C09134=1225.795,-112.726,-36.127,179.386,5.319,149.110
C09135=1225.800,-112.975,-36.117,179.383,5.319,149.111
C09136=1225.805,-113.226,-36.108,179.381,5.319,149.111
C09137=1225.810,-113.475,-36.097,179.379,5.318,149.112
C09138=1225.816,-113.725,-36.087,179.377,5.319,149.113
C09139=1225.821,-113.975,-36.077,179.374,5.318,149.113
C09140=1225.826,-114.224,-36.067,179.372,5.319,149.114
C09141=1225.831,-114.474,-36.057,179.369,5.318,149.115
C09142=1225.837,-114.724,-36.047,179.367,5.318,149.116
C09143=1225.842,-114.974,-36.037,179.365,5.318,149.116
C09144=1225.847,-115.224,-36.027,179.363,5.318,149.117
C09145=1225.853,-115.473,-36.017,179.360,5.318,149.117
C09146=1225.857,-115.723,-36.007,179.358,5.318,149.118
C09147=1225.863,-115.973,-35.997,179.356,5.318,149.119
C09148=1225.869,-116.223,-35.987,179.353,5.318,149.120
C09149=1225.873,-116.472,-35.978,179.351,5.318,149.120
C09150=1225.878,-116.722,-35.967,179.349,5.317,149.121
C09151=1225.884,-116.972,-35.957,179.347,5.318,149.122
C09152=1225.889,-117.221,-35.947,179.344,5.317,149.122
C09153=1225.895,-117.471,-35.938,179.342,5.318,149.123
C09154=1225.900,-117.721,-35.927,179.339,5.317,149.124
C09155=1225.905,-117.971,-35.917,179.337,5.318,149.124
C09156=1225.910,-118.220,-35.907,179.335,5.317,149.125
C09157=1225.915,-118.470,-35.898,179.333,5.317,149.126
C09158=1225.920,-118.720,-35.888,179.331,5.318,149.126
C09159=1225.926,-118.970,-35.878,179.328,5.317,149.127
C09160=1225.931,-119.219,-35.868,179.326,5.318,149.128
C09161=1225.937,-119.469,-35.858,179.323,5.317,149.128
C09162=1225.942,-119.718,-35.849,179.321,5.318,149.129
C09163=1225.947,-119.969,-35.838,179.319,5.317,149.130
C09164=1225.953,-120.219,-35.829,179.317,5.317,149.130
C09165=1225.957,-120.468,-35.819,179.314,5.317,149.131
C09166=1225.963,-120.718,-35.809,179.312,5.317,149.132
C09167=1225.968,-120.968,-35.800,179.310,5.317,149.133
C09168=1225.973,-121.218,-35.790,179.307,5.317,149.133
C09169=1225.978,-121.467,-35.780,179.306,5.317,149.134
C09170=1225.984,-121.717,-35.770,179.303,5.317,149.134
C09171=1225.989,-121.966,-35.761,179.301,5.317,149.135
C09172=1225.994,-122.216,-35.751,179.298,5.317,149.136
C09173=1226.000,-122.467,-35.741,179.296,5.317,149.137
C09174=1226.005,-122.716,-35.731,179.294,5.317,149.137
C09175=1226.010,-122.966,-35.721,179.292,5.317,149.138
C09176=1226.015,-123.215,-35.712,179.289,5.316,149.139
C09177=1226.021,-123.465,-35.702,179.287,5.317,149.139
C09178=1226.026,-123.716,-35.693,179.285,5.317,149.140
C09179=1226.031,-123.965,-35.682,179.282,5.317,149.141
C09180=1226.036,-124.214,-35.673,179.280,5.317,149.141
C09181=1226.042,-124.464,-35.663,179.278,5.316,149.142
C09182=1226.047,-124.714,-35.654,179.276,5.317,149.143
C09183=1226.053,-124.964,-35.644,179.273,5.316,149.143
C09184=1226.058,-125.213,-35.634,179.271,5.316,149.144
C09185=1226.063,-125.464,-35.625,179.269,5.316,149.145
C09186=1226.068,-125.713,-35.615,179.267,5.316,149.145
C09187=1226.074,-125.963,-35.606,179.264,5.316,149.146
C09188=1226.078,-126.213,-35.596,179.262,5.316,149.147
C09189=1225.657,-126.223,-35.632,179.258,5.320,149.149
C09190=1225.652,-125.973,-35.641,179.260,5.319,149.148
C09191=1225.646,-125.724,-35.651,179.263,5.320,149.147
C09192=1225.641,-125.474,-35.660,179.265,5.319,149.147
C09193=1225.636,-125.224,-35.671,179.267,5.320,149.146
C09194=1225.631,-124.975,-35.680,179.269,5.320,149.145
C09195=1225.625,-124.724,-35.690,179.272,5.320,149.145
C09196=1225.620,-124.475,-35.700,179.274,5.320,149.144
C09197=1225.614,-124.225,-35.709,179.276,5.320,149.143
C09198=1225.609,-123.976,-35.719,179.279,5.320,149.143
C09199=1225.603,-123.726,-35.728,179.281,5.319,149.142
C09200=1225.599,-123.476,-35.738,179.283,5.320,149.141
C09201=1225.594,-123.226,-35.748,179.285,5.320,149.141
C09202=1225.588,-122.976,-35.757,179.288,5.320,149.140
C09203=1225.583,-122.727,-35.767,179.290,5.320,149.139
C09204=1225.578,-122.477,-35.776,179.292,5.320,149.138
C09205=1225.572,-122.227,-35.787,179.294,5.320,149.138
C09206=1225.568,-121.977,-35.797,179.297,5.321,149.137
C09207=1225.562,-121.727,-35.806,179.299,5.320,149.137
C09208=1225.557,-121.478,-35.816,179.301,5.321,149.136
C09209=1225.551,-121.229,-35.826,179.304,5.320,149.135
C09210=1225.546,-120.979,-35.835,179.306,5.320,149.134
C09211=1225.541,-120.728,-35.845,179.308,5.321,149.134
C09212=1225.536,-120.479,-35.856,179.310,5.320,149.133
C09213=1225.531,-120.229,-35.864,179.313,5.321,149.132
C09214=1225.525,-119.979,-35.875,179.315,5.320,149.132
C09215=1225.520,-119.730,-35.884,179.317,5.321,149.131
C09216=1225.515,-119.479,-35.894,179.319,5.320,149.130
C09217=1225.510,-119.230,-35.904,179.322,5.321,149.130
C09218=1225.504,-118.981,-35.914,179.324,5.321,149.129
C09219=1225.499,-118.731,-35.924,179.326,5.320,149.128
C09220=1225.494,-118.481,-35.933,179.328,5.321,149.128
C09221=1225.489,-118.231,-35.944,179.331,5.320,149.127
C09222=1225.484,-117.982,-35.953,179.333,5.321,149.126
C09223=1225.478,-117.732,-35.963,179.335,5.321,149.126
C09224=1225.473,-117.481,-35.973,179.338,5.321,149.125
C09225=1225.468,-117.232,-35.983,179.340,5.321,149.124
C09226=1225.462,-116.983,-35.993,179.342,5.321,149.124
C09227=1225.457,-116.733,-36.003,179.344,5.321,149.123
C09228=1225.452,-116.482,-36.013,179.347,5.321,149.122
C09229=1225.447,-116.233,-36.023,179.349,5.321,149.122
C09230=1225.442,-115.984,-36.032,179.351,5.322,149.121
C09231=1225.436,-115.734,-36.043,179.353,5.321,149.120
C09232=1225.431,-115.484,-36.053,179.356,5.321,149.120
C09233=1225.426,-115.234,-36.062,179.358,5.322,149.119
C09234=1225.420,-114.985,-36.072,179.360,5.321,149.118
C09235=1225.415,-114.735,-36.083,179.363,5.322,149.117
C09236=1225.410,-114.485,-36.093,179.365,5.321,149.117
C09237=1225.405,-114.235,-36.103,179.367,5.322,149.116
C09238=1225.399,-113.985,-36.112,179.369,5.322,149.116
C09239=1225.394,-113.735,-36.123,179.372,5.322,149.115
C09240=1225.389,-113.486,-36.132,179.374,5.322,149.114
C09241=1225.384,-113.236,-36.143,179.377,5.322,149.113
C09242=1225.378,-112.987,-36.153,179.379,5.322,149.113
C09243=1225.374,-112.737,-36.163,179.382,5.322,149.112
C09244=1225.368,-112.487,-36.173,179.383,5.322,149.111
C09245=1225.362,-112.238,-36.183,179.385,5.322,149.111
C09246=1225.357,-111.987,-36.193,179.388,5.322,149.110
C09247=1225.352,-111.738,-36.203,179.390,5.322,149.109
C09248=1225.347,-111.488,-36.213,179.393,5.322,149.109
C09249=1225.342,-111.238,-36.223,179.395,5.322,149.108
C09250=1225.336,-110.988,-36.234,179.398,5.322,149.107
C09251=1225.331,-110.739,-36.243,179.399,5.322,149.107
C09252=1225.326,-110.489,-36.254,179.402,5.323,149.106
C09253=1225.321,-110.239,-36.264,179.404,5.322,149.105
C09254=1225.315,-109.990,-36.274,179.407,5.323,149.105
C09255=1225.311,-109.740,-36.284,179.409,5.322,149.104
C09256=1225.305,-109.490,-36.294,179.411,5.323,149.103
C09257=1225.300,-109.241,-36.305,179.413,5.323,149.102
C09258=1225.295,-108.990,-36.315,179.416,5.322,149.102
C09259=1225.289,-108.741,-36.325,179.418,5.323,149.101
C09260=1225.284,-108.492,-36.335,179.420,5.323,149.100
C09261=1225.279,-108.241,-36.346,179.422,5.323,149.100
C09262=1225.274,-107.992,-36.356,179.425,5.323,149.099
C09263=1225.268,-107.742,-36.366,179.427,5.323,149.098
C09264=1225.263,-107.492,-36.377,179.429,5.323,149.098
C09265=1225.258,-107.243,-36.386,179.432,5.323,149.097
C09266=1225.253,-106.993,-36.397,179.434,5.323,149.096
C09267=1225.247,-106.743,-36.407,179.436,5.324,149.096
C09268=1225.242,-106.494,-36.417,179.438,5.323,149.095
C09269=1225.237,-106.243,-36.428,179.441,5.324,149.094
C09270=1225.231,-105.994,-36.438,179.443,5.323,149.094
C09271=1225.226,-105.745,-36.448,179.446,5.324,149.093
C09272=1225.221,-105.494,-36.458,179.448,5.323,149.092
C09273=1225.216,-105.245,-36.468,179.451,5.324,149.091
C09274=1225.211,-104.995,-36.479,179.453,5.323,149.091
C09275=1225.205,-104.745,-36.489,179.455,5.323,149.090
C09276=1225.200,-104.496,-36.500,179.457,5.324,149.090
C09277=1225.195,-104.246,-36.511,179.459,5.323,149.089
C09278=1225.189,-103.996,-36.521,179.462,5.324,149.088
C09279=1225.185,-103.746,-36.531,179.464,5.324,149.087
C09280=1225.179,-103.497,-36.541,179.466,5.324,149.087
C09281=1225.174,-103.247,-36.552,179.469,5.324,149.086
C09282=1225.169,-102.997,-36.562,179.471,5.324,149.085
C09283=1225.163,-102.747,-36.572,179.473,5.324,149.085
C09284=1225.159,-102.498,-36.583,179.476,5.324,149.084
C09285=1225.153,-102.248,-36.594,179.478,5.324,149.083
C09286=1225.148,-101.998,-36.604,179.480,5.325,149.083
C09287=1225.142,-101.748,-36.614,179.482,5.324,149.082
C09288=1225.137,-101.498,-36.625,179.485,5.325,149.081
C09289=1225.133,-101.249,-36.635,179.487,5.324,149.080
C09290=1225.127,-100.978,-36.647,179.490,5.325,149.080
C09291=1225.121,-100.706,-36.658,179.492,5.324,149.079
C09292=1225.115,-100.436,-36.669,179.495,5.324,149.078
C09293=1225.110,-100.165,-36.681,179.498,5.325,149.077
C09294=1225.104,-99.915,-36.691,179.500,5.324,149.077
C09295=1225.099,-99.665,-36.702,179.503,5.325,149.076
C09296=1225.093,-99.416,-36.712,179.504,5.325,149.075
C09297=1225.089,-99.166,-36.723,179.507,5.325,149.075
C09298=1225.084,-98.917,-36.733,179.509,5.325,149.074
C09299=1225.079,-98.666,-36.744,179.512,5.325,149.073
C09300=1225.074,-98.418,-36.755,179.514,5.325,149.073
C09301=1225.069,-98.167,-36.765,179.516,5.325,149.072
C09302=1225.063,-97.918,-36.775,179.518,5.325,149.071
C09303=1225.058,-97.667,-36.786,179.521,5.325,149.070
C09304=1225.053,-97.419,-36.797,179.523,5.325,149.070
C09305=1225.047,-97.168,-36.808,179.525,5.325,149.069
C09306=1225.041,-96.918,-36.818,179.527,5.326,149.069
C09307=1225.037,-96.669,-36.830,179.530,5.325,149.068
C09308=1225.031,-96.419,-36.840,179.532,5.326,149.067
C09309=1225.026,-96.169,-36.850,179.534,5.325,149.066
C09310=1225.020,-95.919,-36.861,179.537,5.326,149.066
C09311=1225.016,-95.670,-36.872,179.539,5.325,149.065
C09312=1225.010,-95.420,-36.882,179.542,5.326,149.064
C09313=1225.005,-95.171,-36.893,179.544,5.326,149.064
C09314=1225.000,-94.921,-36.904,179.547,5.326,149.063
C09315=1224.995,-94.671,-36.914,179.549,5.326,149.062
C09316=1224.990,-94.421,-36.925,179.551,5.326,149.061
C09317=1224.985,-94.172,-36.936,179.553,5.326,149.061
C09318=1224.980,-93.921,-36.946,179.556,5.326,149.060
C09319=1224.974,-93.673,-36.957,179.558,5.326,149.060
C09320=1224.969,-93.422,-36.968,179.560,5.327,149.059
C09321=1224.963,-93.173,-36.979,179.562,5.326,149.058
C09322=1224.958,-92.923,-36.990,179.565,5.327,149.057
C09323=1224.953,-92.673,-37.000,179.567,5.326,149.057
C09324=1224.948,-92.424,-37.011,179.570,5.327,149.056
C09325=1224.943,-92.173,-37.022,179.572,5.326,149.055
C09326=1224.938,-91.924,-37.033,179.575,5.327,149.055
C09327=1224.933,-91.674,-37.043,179.577,5.326,149.054
C09328=1224.927,-91.425,-37.054,179.579,5.327,149.053
C09329=1224.922,-91.175,-37.065,179.582,5.327,149.052
C09330=1224.916,-90.926,-37.076,179.584,5.327,149.052
C09331=1224.911,-90.676,-37.087,179.586,5.327,149.051
C09332=1224.906,-90.425,-37.098,179.588,5.327,149.051
C09333=1224.901,-90.176,-37.108,179.591,5.327,149.050
C09334=1224.896,-89.926,-37.119,179.593,5.328,149.049
C09335=1224.891,-89.677,-37.130,179.595,5.327,149.048
C09336=1224.885,-89.427,-37.141,179.598,5.328,149.048
C09337=1224.880,-89.177,-37.152,179.600,5.327,149.047
C09338=1224.875,-88.928,-37.163,179.603,5.328,149.046
C09339=1224.870,-88.678,-37.174,179.605,5.327,149.046
C09340=1224.865,-88.428,-37.185,179.608,5.328,149.045
C09341=1224.860,-88.179,-37.195,179.610,5.327,149.044
C09342=1224.854,-87.929,-37.207,179.612,5.328,149.043
C09343=1224.849,-87.679,-37.217,179.614,5.328,149.043
C09344=1224.844,-87.430,-37.229,179.617,5.328,149.042
C09345=1224.839,-87.179,-37.239,179.619,5.328,149.041
C09346=1224.833,-86.930,-37.251,179.621,5.328,149.041
C09347=1224.828,-86.681,-37.262,179.623,5.328,149.040
C09348=1224.823,-86.430,-37.273,179.626,5.329,149.039
C09349=1224.818,-86.181,-37.284,179.628,5.328,149.039
C09350=1224.813,-85.931,-37.294,179.631,5.329,149.038
C09351=1224.808,-85.681,-37.306,179.633,5.328,149.037
C09352=1224.802,-85.432,-37.317,179.636,5.329,149.037
C09353=1224.797,-85.182,-37.328,179.638,5.328,149.036
C09354=1224.793,-84.932,-37.339,179.640,5.329,149.035
C09355=1224.786,-84.683,-37.350,179.642,5.328,149.034
C09356=1224.782,-84.433,-37.361,179.645,5.329,149.034
C09357=1224.777,-84.183,-37.372,179.647,5.329,149.033
C09358=1224.771,-83.934,-37.382,179.650,5.329,149.032
C09359=1224.766,-83.684,-37.394,179.652,5.329,149.032
C09360=1224.761,-83.434,-37.406,179.655,5.329,149.031
C09361=1224.756,-83.185,-37.416,179.657,5.329,149.030
C09362=1224.750,-82.935,-37.428,179.659,5.329,149.029
C09363=1224.745,-82.685,-37.439,179.662,5.329,149.029
C09364=1224.741,-82.435,-37.450,179.664,5.330,149.028
C09365=1224.734,-82.186,-37.461,179.666,5.330,149.028
C09366=1224.730,-81.936,-37.472,179.668,5.330,149.027
C09367=1224.725,-81.686,-37.484,179.671,5.330,149.026
C09368=1224.719,-81.436,-37.495,179.673,5.330,149.025
C09369=1224.714,-81.187,-37.506,179.676,5.330,149.025
C09370=1224.709,-80.937,-37.517,179.678,5.330,149.024
C09371=1224.704,-80.687,-37.529,179.681,5.330,149.023
C09372=1224.698,-80.438,-37.539,179.683,5.330,149.023
C09373=1224.694,-80.188,-37.550,179.685,5.330,149.022
C09374=1224.688,-79.938,-37.562,179.688,5.330,149.021
C09375=1224.683,-79.689,-37.573,179.690,5.331,149.020
C09376=1224.678,-79.440,-37.585,179.692,5.330,149.020
C09377=1224.672,-79.189,-37.596,179.695,5.331,149.019
C09378=1224.668,-78.939,-37.607,179.697,5.330,149.018
C09379=1224.663,-78.691,-37.618,179.700,5.331,149.018
C09380=1224.657,-78.441,-37.630,179.702,5.330,149.017
C09381=1224.652,-78.191,-37.641,179.704,5.331,149.016
C09382=1224.647,-77.940,-37.652,179.707,5.331,149.015
C09383=1224.642,-77.691,-37.664,179.709,5.331,149.015
C09384=1224.637,-77.442,-37.675,179.711,5.331,149.014
C09385=1224.631,-77.192,-37.686,179.713,5.331,149.014
C09386=1224.627,-76.942,-37.698,179.716,5.331,149.013
C09387=1224.621,-76.692,-37.710,179.718,5.332,149.012
C09388=1224.616,-76.443,-37.721,179.721,5.332,149.011
C09389=1224.610,-76.193,-37.732,179.723,5.332,149.011
C09390=1224.605,-75.943,-37.743,179.726,5.332,149.010
C09391=1224.600,-75.693,-37.755,179.728,5.332,149.009
C09392=1224.595,-75.444,-37.766,179.730,5.332,149.009
C09393=1224.590,-75.195,-37.777,179.733,5.332,149.008
C09394=1224.584,-74.924,-37.789,179.735,5.332,149.007
C09395=1224.579,-74.653,-37.802,179.738,5.332,149.006
C09396=1224.573,-74.383,-37.814,179.740,5.332,149.006
C09397=1224.568,-74.113,-37.827,179.743,5.333,149.005
C09398=1224.562,-73.863,-37.839,179.745,5.332,149.004
C09399=1224.557,-73.614,-37.850,179.748,5.333,149.003
C09400=1224.551,-73.364,-37.862,179.750,5.332,149.003
C09401=1224.547,-73.114,-37.873,179.753,5.333,149.002
C09402=1224.541,-72.864,-37.885,179.755,5.332,149.001
C09403=1224.537,-72.615,-37.896,179.757,5.333,149.001
C09404=1224.531,-72.365,-37.908,179.760,5.333,149.000
C09405=1224.526,-72.116,-37.919,179.762,5.333,148.999
C09406=1224.520,-71.866,-37.931,179.765,5.333,148.998
C09407=1224.516,-71.616,-37.942,179.767,5.333,148.998
C09408=1224.510,-71.366,-37.954,179.770,5.334,148.997
C09409=1224.506,-71.117,-37.965,179.772,5.333,148.996
C09410=1224.500,-70.867,-37.977,179.774,5.334,148.996
C09411=1224.495,-70.618,-37.988,179.776,5.333,148.995
C09412=1224.489,-70.368,-38.000,179.779,5.334,148.994
C09413=1224.485,-70.118,-38.011,179.781,5.334,148.994
C09414=1224.479,-69.868,-38.023,179.783,5.334,148.993
C09415=1224.474,-69.619,-38.035,179.785,5.334,148.992
C09416=1224.469,-69.369,-38.047,179.788,5.334,148.992
C09417=1224.464,-69.119,-38.058,179.791,5.335,148.991
C09418=1224.459,-68.869,-38.070,179.793,5.335,148.990
C09419=1224.453,-68.620,-38.081,179.796,5.335,148.989
C09420=1224.448,-68.370,-38.093,179.798,5.335,148.989
C09421=1224.443,-68.121,-38.104,179.800,5.335,148.988
C09422=1224.438,-67.871,-38.116,179.802,5.335,148.987
C09423=1224.433,-67.622,-38.128,179.805,5.335,148.987
C09424=1224.428,-67.372,-38.140,179.807,5.335,148.986
C09425=1224.422,-67.122,-38.152,179.810,5.335,148.985
C09426=1224.418,-66.872,-38.163,179.812,5.335,148.985
C09427=1224.412,-66.622,-38.175,179.815,5.335,148.984
C09428=1224.407,-66.373,-38.187,179.817,5.336,148.983
C09429=1224.401,-66.123,-38.198,179.819,5.336,148.982
C09430=1224.396,-65.874,-38.211,179.822,5.336,148.982
C09431=1224.392,-65.624,-38.222,179.824,5.336,148.981
C09432=1224.386,-65.374,-38.234,179.827,5.336,148.980
C09433=1224.381,-65.125,-38.246,179.829,5.336,148.980
C09434=1224.376,-64.875,-38.257,179.832,5.336,148.979
C09435=1224.371,-64.626,-38.270,179.834,5.336,148.978
C09436=1224.366,-64.376,-38.281,179.836,5.336,148.977
C09437=1224.361,-64.126,-38.293,179.839,5.337,148.977
C09438=1224.355,-63.876,-38.305,179.841,5.337,148.976
C09439=1224.350,-63.626,-38.317,179.844,5.337,148.975
C09440=1224.346,-63.377,-38.329,179.846,5.337,148.975
C09441=1224.340,-63.127,-38.340,179.848,5.337,148.974
C09442=1224.335,-62.877,-38.352,179.851,5.337,148.973
C09443=1224.329,-62.627,-38.364,179.853,5.337,148.973
C09444=1224.325,-62.378,-38.376,179.855,5.337,148.972
C09445=1224.319,-62.128,-38.388,179.858,5.337,148.971
C09446=1224.314,-61.878,-38.400,179.861,5.338,148.970
C09447=1224.309,-61.629,-38.411,179.863,5.337,148.970
C09448=1224.304,-61.379,-38.424,179.865,5.338,148.969
C09449=1224.299,-61.130,-38.436,179.867,5.338,148.968
C09450=1224.293,-60.880,-38.448,179.870,5.338,148.968
C09451=1224.289,-60.631,-38.460,179.872,5.338,148.967
C09452=1224.284,-60.381,-38.472,179.875,5.338,148.966
C09453=1224.278,-60.131,-38.483,179.878,5.339,148.965
C09454=1224.273,-59.881,-38.496,179.879,5.339,148.965
C09455=1224.268,-59.632,-38.507,179.882,5.339,148.964
C09456=1224.263,-59.382,-38.519,179.884,5.339,148.964
C09457=1224.258,-59.133,-38.532,179.887,5.339,148.963
C09458=1224.252,-58.883,-38.544,179.889,5.339,148.962
C09459=1224.247,-58.633,-38.556,179.891,5.339,148.961
C09460=1224.242,-58.384,-38.568,179.894,5.340,148.961
C09461=1224.237,-58.134,-38.579,179.896,5.340,148.960
C09462=1224.232,-57.884,-38.592,179.899,5.340,148.959
C09463=1224.227,-57.634,-38.604,179.901,5.340,148.959
C09464=1224.221,-57.385,-38.616,179.904,5.340,148.958
C09465=1224.217,-57.136,-38.628,179.906,5.340,148.957
C09466=1224.211,-56.886,-38.640,179.908,5.340,148.957
C09467=1224.206,-56.636,-38.652,179.911,5.341,148.956
C09468=1224.201,-56.386,-38.664,179.913,5.340,148.955
C09469=1224.196,-56.137,-38.677,179.916,5.341,148.954
C09470=1224.190,-55.887,-38.689,179.918,5.341,148.954
C09471=1224.186,-55.638,-38.701,179.920,5.341,148.953
C09472=1224.180,-55.388,-38.713,179.923,5.341,148.952
C09473=1224.175,-55.139,-38.725,179.925,5.341,148.952
C09474=1224.170,-54.888,-38.737,179.928,5.342,148.951
C09475=1224.165,-54.638,-38.749,179.930,5.341,148.950
C09476=1224.160,-54.389,-38.762,179.933,5.342,148.950
C09477=1224.154,-54.139,-38.774,179.935,5.341,148.949
C09478=1224.150,-53.890,-38.786,179.937,5.342,148.948
C09479=1224.145,-53.641,-38.798,179.939,5.342,148.947
C09480=1224.139,-53.391,-38.810,179.942,5.342,148.947
C09481=1224.134,-53.141,-38.823,179.945,5.343,148.946
C09482=1224.129,-52.891,-38.835,179.947,5.342,148.945
C09483=1224.124,-52.642,-38.847,179.950,5.343,148.945
C09484=1224.119,-52.392,-38.860,179.952,5.342,148.944
C09485=1224.114,-52.142,-38.872,179.954,5.343,148.943
C09486=1224.108,-51.892,-38.884,179.957,5.343,148.942
C09487=1224.103,-51.643,-38.897,179.959,5.343,148.942
C09488=1224.098,-51.394,-38.909,179.962,5.343,148.941
C09489=1224.093,-51.144,-38.921,179.964,5.343,148.940
C09490=1224.088,-50.895,-38.933,179.966,5.344,148.940
C09491=1224.083,-50.645,-38.945,179.969,5.344,148.939
C09492=1224.078,-50.395,-38.958,179.971,5.344,148.938
C09493=1224.073,-50.145,-38.971,179.974,5.344,148.938
C09494=1224.068,-49.895,-38.983,179.976,5.344,148.937
C09495=1224.063,-49.646,-38.995,179.979,5.344,148.936
C09496=1224.057,-49.396,-39.007,179.981,5.345,148.935
C09497=1224.052,-49.147,-39.020,179.983,5.345,148.935
C09498=1224.046,-48.877,-39.034,179.986,5.345,148.934
C09499=1224.041,-48.607,-39.047,179.989,5.345,148.933
C09500=1224.036,-48.337,-39.060,179.991,5.345,148.932
C09501=1224.030,-48.067,-39.073,179.994,5.345,148.932
C09502=1224.025,-47.818,-39.086,179.997,5.346,148.931
C09503=1224.020,-47.569,-39.098,179.999,5.345,148.930
C09504=1224.015,-47.319,-39.111,-179.999,5.346,148.930
C09505=1224.010,-47.069,-39.123,-179.997,5.346,148.929
C09506=1224.004,-46.819,-39.136,-179.994,5.346,148.928
C09507=1223.999,-46.570,-39.149,-179.991,5.347,148.927
C09508=1223.994,-46.320,-39.161,-179.989,5.346,148.927
C09509=1223.988,-46.070,-39.173,-179.986,5.347,148.926
C09510=1223.984,-45.820,-39.186,-179.984,5.346,148.925
C09511=1223.979,-45.571,-39.199,-179.982,5.347,148.925
C09512=1223.973,-45.321,-39.211,-179.979,5.347,148.924
C09513=1223.968,-45.072,-39.224,-179.977,5.347,148.923
C09514=1223.963,-44.822,-39.236,-179.974,5.347,148.923
C09515=1223.959,-44.572,-39.249,-179.972,5.347,148.922
C09516=1223.953,-44.322,-39.261,-179.970,5.348,148.921
C09517=1223.948,-44.073,-39.274,-179.967,5.348,148.920
C09518=1223.943,-43.824,-39.286,-179.965,5.348,148.920
C09519=1223.938,-43.575,-39.299,-179.962,5.348,148.919
C09520=1223.933,-43.324,-39.312,-179.960,5.348,148.918
C09521=1223.927,-43.075,-39.325,-179.957,5.348,148.918
C09522=1223.922,-42.825,-39.337,-179.955,5.349,148.917
C09523=1223.917,-42.576,-39.349,-179.953,5.349,148.916
C09524=1223.912,-42.326,-39.362,-179.950,5.349,148.916
C09525=1223.907,-42.076,-39.375,-179.947,5.350,148.915
C09526=1223.902,-41.827,-39.388,-179.945,5.349,148.914
C09527=1223.896,-41.577,-39.401,-179.943,5.350,148.913
C09528=1223.891,-41.327,-39.413,-179.940,5.349,148.913
C09529=1223.886,-41.077,-39.426,-179.938,5.350,148.912
C09530=1223.881,-40.828,-39.438,-179.935,5.350,148.911
C09531=1223.877,-40.578,-39.451,-179.933,5.350,148.911
C09532=1223.872,-40.329,-39.464,-179.930,5.350,148.910
C09533=1223.866,-40.079,-39.476,-179.928,5.351,148.909
C09534=1223.861,-39.830,-39.490,-179.926,5.351,148.909
C09535=1223.856,-39.580,-39.503,-179.923,5.351,148.908
C09536=1223.851,-39.330,-39.515,-179.921,5.351,148.907
C09537=1223.846,-39.081,-39.528,-179.918,5.351,148.906
C09538=1223.841,-38.831,-39.541,-179.916,5.352,148.906
C09539=1223.835,-38.581,-39.554,-179.913,5.351,148.905
C09540=1223.830,-38.332,-39.567,-179.911,5.352,148.904
C09541=1223.825,-38.083,-39.579,-179.909,5.352,148.904
C09542=1223.820,-37.832,-39.591,-179.906,5.352,148.903
C09543=1223.814,-37.583,-39.605,-179.903,5.353,148.902
C09544=1223.809,-37.333,-39.617,-179.901,5.352,148.902
C09545=1223.805,-37.083,-39.630,-179.899,5.353,148.901
C09546=1223.800,-36.834,-39.643,-179.896,5.353,148.900
C09547=1223.794,-36.584,-39.656,-179.894,5.353,148.899
C09548=1223.790,-36.335,-39.670,-179.891,5.353,148.899
C09549=1223.784,-36.086,-39.682,-179.889,5.354,148.898
C09550=1223.779,-35.836,-39.695,-179.887,5.354,148.897
C09551=1223.774,-35.586,-39.708,-179.884,5.354,148.897
C09552=1223.769,-35.337,-39.721,-179.882,5.354,148.896
C09553=1223.764,-35.087,-39.734,-179.879,5.354,148.895
C09554=1223.759,-34.837,-39.747,-179.876,5.355,148.895
C09555=1223.753,-34.588,-39.760,-179.874,5.354,148.894
C09556=1223.748,-34.338,-39.772,-179.872,5.355,148.893
C09557=1223.744,-34.088,-39.785,-179.869,5.355,148.892
C09558=1223.738,-33.839,-39.799,-179.867,5.355,148.892
C09559=1223.733,-33.589,-39.811,-179.864,5.356,148.891
C09560=1223.728,-33.339,-39.824,-179.862,5.356,148.890
C09561=1223.722,-33.090,-39.837,-179.860,5.356,148.890
C09562=1223.718,-32.840,-39.851,-179.857,5.356,148.889
C09563=1223.713,-32.591,-39.864,-179.855,5.356,148.888
C09564=1223.707,-32.341,-39.877,-179.852,5.356,148.888
C09565=1223.703,-32.091,-39.890,-179.849,5.357,148.887
C09566=1223.698,-31.842,-39.902,-179.847,5.357,148.886
C09567=1223.692,-31.592,-39.916,-179.845,5.357,148.885
C09568=1223.687,-31.342,-39.928,-179.842,5.358,148.885
C09569=1223.682,-31.094,-39.942,-179.840,5.357,148.884
C09570=1223.677,-30.843,-39.955,-179.837,5.358,148.883
C09571=1223.672,-30.594,-39.968,-179.835,5.358,148.883
C09572=1223.667,-30.344,-39.982,-179.833,5.358,148.882
C09573=1223.662,-30.094,-39.994,-179.830,5.358,148.881
C09574=1223.657,-29.846,-40.007,-179.827,5.359,148.881
C09575=1223.652,-29.595,-40.021,-179.825,5.359,148.880
C09576=1223.646,-29.346,-40.034,-179.823,5.359,148.879
C09577=1223.641,-29.096,-40.047,-179.820,5.360,148.878
C09578=1223.636,-28.847,-40.060,-179.818,5.359,148.878
C09579=1223.632,-28.597,-40.073,-179.815,5.360,148.877
C09580=1223.626,-28.347,-40.087,-179.812,5.360,148.876
C09581=1223.621,-28.098,-40.099,-179.810,5.360,148.876
C09582=1223.616,-27.848,-40.114,-179.808,5.360,148.875
C09583=1223.611,-27.599,-40.126,-179.806,5.360,148.874
C09584=1223.605,-27.349,-40.140,-179.803,5.361,148.874
C09585=1223.601,-27.100,-40.153,-179.800,5.361,148.873
C09586=1223.596,-26.850,-40.166,-179.798,5.361,148.872
C09587=1223.590,-26.600,-40.179,-179.796,5.361,148.872
C09588=1223.586,-26.350,-40.192,-179.793,5.362,148.871
C09589=1223.580,-26.101,-40.206,-179.791,5.361,148.870
C09590=1223.576,-25.851,-40.219,-179.788,5.362,148.869
C09591=1223.570,-25.602,-40.232,-179.786,5.362,148.869
C09592=1223.566,-25.352,-40.246,-179.783,5.362,148.868
C09593=1223.560,-25.103,-40.259,-179.781,5.363,148.867
C09594=1223.556,-24.853,-40.273,-179.778,5.363,148.867
C09595=1223.550,-24.604,-40.286,-179.777,5.363,148.866
C09596=1223.545,-24.354,-40.299,-179.774,5.364,148.865
C09597=1223.540,-24.105,-40.313,-179.771,5.364,148.865
C09598=1223.535,-23.855,-40.326,-179.769,5.364,148.864
C09599=1223.529,-23.605,-40.339,-179.766,5.364,148.863
C09600=1223.525,-23.356,-40.353,-179.764,5.365,148.863
C09601=1223.519,-23.106,-40.366,-179.762,5.365,148.862
C09602=1223.514,-22.837,-40.381,-179.759,5.365,148.861
C09603=1223.509,-22.567,-40.395,-179.756,5.365,148.860
C09604=1223.503,-22.298,-40.409,-179.753,5.366,148.860
C09605=1223.497,-22.029,-40.424,-179.751,5.366,148.859
C09606=1223.493,-21.779,-40.437,-179.749,5.366,148.858
C09607=1223.487,-21.530,-40.451,-179.746,5.366,148.858
C09608=1223.483,-21.280,-40.464,-179.743,5.367,148.857
C09609=1223.477,-21.031,-40.478,-179.741,5.367,148.856
C09610=1223.472,-20.780,-40.491,-179.738,5.367,148.856
C09611=1223.467,-20.532,-40.505,-179.736,5.368,148.855
C09612=1223.462,-20.281,-40.518,-179.734,5.367,148.854
C09613=1223.457,-20.033,-40.532,-179.731,5.368,148.853
C09614=1223.452,-19.782,-40.545,-179.728,5.368,148.853
C09615=1223.447,-19.533,-40.560,-179.726,5.369,148.852
C09616=1223.442,-19.283,-40.572,-179.724,5.368,148.851
C09617=1223.437,-19.033,-40.586,-179.721,5.369,148.851
C09618=1223.431,-18.784,-40.600,-179.718,5.369,148.850
C09619=1223.427,-18.534,-40.613,-179.716,5.369,148.849
C09620=1223.421,-18.285,-40.627,-179.714,5.370,148.849
C09621=1223.416,-18.035,-40.641,-179.711,5.370,148.848
C09622=1223.412,-17.786,-40.654,-179.709,5.370,148.847
C09623=1223.406,-17.536,-40.668,-179.706,5.370,148.846
C09624=1223.401,-17.287,-40.681,-179.704,5.371,148.846
C09625=1223.396,-17.038,-40.695,-179.701,5.371,148.845
C09626=1223.391,-16.787,-40.709,-179.699,5.371,148.844
C09627=1223.386,-16.538,-40.723,-179.696,5.372,148.844
C09628=1223.381,-16.288,-40.736,-179.693,5.372,148.843
C09629=1223.376,-16.039,-40.750,-179.691,5.372,148.842
C09630=1223.370,-15.790,-40.764,-179.689,5.372,148.842
C09631=1223.366,-15.540,-40.777,-179.686,5.373,148.841
C09632=1223.361,-15.290,-40.791,-179.684,5.372,148.840
C09633=1223.355,-15.041,-40.805,-179.681,5.373,148.840
C09634=1223.350,-14.791,-40.818,-179.679,5.373,148.839
C09635=1223.346,-14.541,-40.832,-179.677,5.373,148.838
C09636=1223.340,-14.292,-40.846,-179.674,5.374,148.837
C09637=1223.335,-14.042,-40.860,-179.671,5.374,148.837
C09638=1223.330,-13.792,-40.873,-179.669,5.375,148.836
C09639=1223.325,-13.543,-40.887,-179.667,5.374,148.835
C09640=1223.320,-13.293,-40.901,-179.664,5.375,148.835
C09641=1223.315,-13.043,-40.915,-179.661,5.375,148.834
C09642=1223.310,-12.795,-40.928,-179.659,5.375,148.833
C09643=1223.305,-12.545,-40.943,-179.657,5.376,148.833
C09644=1223.300,-12.295,-40.956,-179.654,5.376,148.832
C09645=1223.294,-12.046,-40.970,-179.651,5.377,148.831
C09646=1223.290,-11.796,-40.984,-179.649,5.376,148.831
C09647=1223.285,-11.546,-40.998,-179.646,5.377,148.830
C09648=1223.279,-11.297,-41.011,-179.644,5.377,148.829
C09649=1223.274,-11.047,-41.026,-179.642,5.377,148.828
C09650=1223.269,-10.797,-41.040,-179.639,5.378,148.828
C09651=1223.264,-10.549,-41.053,-179.636,5.378,148.827
C09652=1223.259,-10.299,-41.068,-179.634,5.379,148.826
C09653=1223.254,-10.049,-41.081,-179.632,5.378,148.826
C09654=1223.249,-9.800,-41.095,-179.629,5.379,148.825
C09655=1223.244,-9.550,-41.109,-179.626,5.379,148.824
C09656=1223.239,-9.301,-41.123,-179.624,5.379,148.824
C09657=1223.234,-9.051,-41.137,-179.622,5.380,148.823
C09658=1223.229,-8.802,-41.151,-179.619,5.380,148.822
C09659=1223.224,-8.552,-41.165,-179.616,5.381,148.822
C09660=1223.219,-8.302,-41.179,-179.614,5.380,148.821
C09661=1223.213,-8.053,-41.193,-179.612,5.381,148.820
C09662=1223.208,-7.803,-41.207,-179.609,5.381,148.819
C09663=1223.204,-7.554,-41.221,-179.607,5.381,148.819
C09664=1223.199,-7.304,-41.235,-179.604,5.381,148.818
C09665=1223.193,-7.055,-41.249,-179.602,5.382,148.817
C09666=1223.189,-6.805,-41.263,-179.599,5.383,148.817
C09667=1223.184,-6.556,-41.278,-179.597,5.382,148.816
C09668=1223.179,-6.306,-41.292,-179.594,5.383,148.815
C09669=1223.173,-6.057,-41.306,-179.592,5.384,148.815
C09670=1223.168,-5.807,-41.319,-179.589,5.384,148.814
C09671=1223.163,-5.557,-41.334,-179.587,5.384,148.813
C09672=1223.158,-5.307,-41.348,-179.585,5.384,148.813
C09673=1223.154,-5.058,-41.362,-179.582,5.385,148.812
C09674=1223.148,-4.809,-41.376,-179.579,5.385,148.811
C09675=1223.143,-4.559,-41.390,-179.577,5.385,148.811
C09676=1223.138,-4.309,-41.404,-179.575,5.386,148.810
C09677=1223.133,-4.060,-41.418,-179.572,5.386,148.809
C09678=1223.128,-3.811,-41.432,-179.570,5.386,148.809
C09679=1223.123,-3.561,-41.447,-179.567,5.386,148.808
C09680=1223.118,-3.311,-41.461,-179.565,5.387,148.807
C09681=1223.113,-3.061,-41.475,-179.562,5.387,148.807
C09682=1223.108,-2.812,-41.489,-179.560,5.387,148.806
C09683=1223.102,-2.563,-41.503,-179.557,5.388,148.805
C09684=1223.098,-2.314,-41.518,-179.555,5.388,148.804
C09685=1223.093,-2.064,-41.533,-179.552,5.389,148.804
C09686=1223.088,-1.814,-41.547,-179.550,5.388,148.803
C09687=1223.083,-1.564,-41.561,-179.547,5.389,148.802
C09688=1223.078,-1.315,-41.575,-179.544,5.389,148.802
C09689=1223.072,-1.066,-41.589,-179.542,5.390,148.801
C09690=1223.067,-0.816,-41.604,-179.540,5.390,148.800
C09691=1223.062,-0.566,-41.618,-179.537,5.390,148.800
C09692=1223.057,-0.317,-41.632,-179.534,5.391,148.799
C09693=1223.052,-0.067,-41.646,-179.532,5.391,148.798
C09694=1223.047,0.183,-41.661,-179.530,5.391,148.798
C09695=1223.042,0.431,-41.675,-179.527,5.391,148.797
C09696=1223.037,0.681,-41.690,-179.524,5.392,148.796
C09697=1223.032,0.931,-41.704,-179.522,5.392,148.796
C09698=1223.027,1.180,-41.718,-179.520,5.392,148.795
C09699=1223.022,1.430,-41.733,-179.517,5.393,148.794
C09700=1223.017,1.680,-41.747,-179.514,5.393,148.793
C09701=1223.012,1.929,-41.762,-179.512,5.394,148.793
C09702=1223.007,2.179,-41.777,-179.509,5.394,148.792
C09703=1223.002,2.428,-41.790,-179.507,5.394,148.791
C09704=1222.997,2.678,-41.805,-179.505,5.395,148.791
C09705=1222.992,2.927,-41.819,-179.502,5.395,148.790
C09706=1222.987,3.196,-41.835,-179.499,5.395,148.789
C09707=1222.981,3.465,-41.850,-179.496,5.396,148.789
C09708=1222.976,3.734,-41.867,-179.494,5.396,148.788
C09709=1222.970,4.003,-41.882,-179.492,5.396,148.787
C09710=1222.965,4.252,-41.897,-179.489,5.397,148.787
C09711=1222.961,4.502,-41.911,-179.486,5.397,148.786
C09712=1222.956,4.752,-41.925,-179.484,5.398,148.785
C09713=1222.950,5.001,-41.939,-179.481,5.398,148.785
C09714=1222.945,5.250,-41.955,-179.479,5.398,148.784
C09715=1222.940,5.500,-41.969,-179.476,5.399,148.783
C09716=1222.935,5.750,-41.983,-179.474,5.399,148.782
C09717=1222.930,5.999,-41.998,-179.471,5.400,148.782
C09718=1222.925,6.249,-42.013,-179.469,5.399,148.781
C09719=1222.920,6.498,-42.027,-179.466,5.400,148.780
C09720=1222.915,6.748,-42.042,-179.464,5.400,148.780
C09721=1222.910,6.997,-42.057,-179.461,5.401,148.779
C09722=1222.905,7.247,-42.071,-179.458,5.401,148.778
C09723=1222.900,7.496,-42.086,-179.456,5.401,148.778
C09724=1222.895,7.746,-42.100,-179.454,5.402,148.777
C09725=1222.890,7.996,-42.115,-179.451,5.402,148.776
C09726=1222.885,8.245,-42.130,-179.448,5.403,148.776
C09727=1222.880,8.495,-42.144,-179.446,5.402,148.775
C09728=1222.875,8.744,-42.159,-179.444,5.403,148.774
C09729=1222.870,8.994,-42.174,-179.441,5.404,148.774
C09730=1222.865,9.244,-42.189,-179.439,5.404,148.773
C09731=1222.860,9.493,-42.204,-179.436,5.405,148.772
C09732=1222.855,9.742,-42.218,-179.434,5.405,148.772
C09733=1222.850,9.992,-42.233,-179.431,5.405,148.771
C09734=1222.845,10.241,-42.248,-179.429,5.406,148.770
C09735=1222.840,10.491,-42.263,-179.426,5.406,148.770
C09736=1222.835,10.740,-42.277,-179.423,5.407,148.769
C09737=1222.830,10.990,-42.293,-179.421,5.406,148.768
C09738=1222.825,11.239,-42.307,-179.419,5.407,148.768
C09739=1222.820,11.488,-42.322,-179.416,5.407,148.767
C09740=1222.814,11.738,-42.337,-179.413,5.408,148.766
C09741=1222.810,11.988,-42.352,-179.411,5.408,148.766
C09742=1222.805,12.237,-42.366,-179.409,5.408,148.765
C09743=1222.799,12.487,-42.382,-179.406,5.409,148.764
C09744=1222.794,12.736,-42.396,-179.403,5.409,148.763
C09745=1222.790,12.985,-42.411,-179.401,5.410,148.763
C09746=1222.785,13.235,-42.425,-179.398,5.410,148.762
C09747=1222.779,13.485,-42.441,-179.396,5.410,148.761
C09748=1222.775,13.734,-42.455,-179.394,5.411,148.761
C09749=1222.769,13.984,-42.471,-179.391,5.411,148.760
C09750=1222.764,14.233,-42.485,-179.389,5.412,148.760
C09751=1222.760,14.483,-42.500,-179.386,5.413,148.759
C09752=1222.754,14.732,-42.515,-179.384,5.412,148.758
C09753=1222.749,14.982,-42.530,-179.381,5.413,148.758
C09754=1222.745,15.231,-42.545,-179.379,5.413,148.757
C09755=1222.739,15.481,-42.560,-179.376,5.414,148.756
C09756=1222.734,15.730,-42.575,-179.373,5.414,148.755
C09757=1222.729,15.979,-42.590,-179.371,5.415,148.755
C09758=1222.724,16.230,-42.605,-179.369,5.415,148.754
C09759=1222.720,16.479,-42.620,-179.366,5.415,148.753
C09760=1222.714,16.728,-42.635,-179.363,5.416,148.753
C09761=1222.709,16.978,-42.650,-179.361,5.416,148.752
C09762=1222.704,17.227,-42.665,-179.358,5.417,148.751
C09763=1222.699,17.476,-42.680,-179.356,5.416,148.751
C09764=1222.694,17.726,-42.694,-179.353,5.417,148.750
C09765=1222.689,17.975,-42.710,-179.351,5.418,148.750
C09766=1222.684,18.225,-42.725,-179.348,5.418,148.749
C09767=1222.679,18.475,-42.740,-179.346,5.419,148.748
C09768=1222.675,18.724,-42.755,-179.343,5.420,148.748
C09769=1222.669,18.974,-42.771,-179.341,5.419,148.747
C09770=1222.665,19.223,-42.786,-179.338,5.420,148.746
C09771=1222.659,19.473,-42.801,-179.336,5.420,148.745
C09772=1222.654,19.722,-42.816,-179.333,5.421,148.745
C09773=1222.649,19.971,-42.831,-179.330,5.421,148.744
C09774=1222.644,20.220,-42.846,-179.328,5.422,148.743
C09775=1222.639,20.471,-42.862,-179.326,5.422,148.743
C09776=1222.635,20.720,-42.877,-179.323,5.422,148.742
C09777=1222.629,20.970,-42.892,-179.320,5.423,148.741
C09778=1222.625,21.219,-42.907,-179.318,5.423,148.741
C09779=1222.619,21.469,-42.922,-179.315,5.424,148.740
C09780=1222.614,21.718,-42.937,-179.313,5.425,148.740
C09781=1222.609,21.967,-42.953,-179.311,5.424,148.739
C09782=1222.605,22.217,-42.968,-179.308,5.425,148.738
C09783=1222.599,22.466,-42.984,-179.306,5.425,148.738
C09784=1222.595,22.716,-42.999,-179.303,5.426,148.737
C09785=1222.589,22.966,-43.013,-179.300,5.427,148.736
C09786=1222.584,23.215,-43.028,-179.298,5.427,148.735
C09787=1222.580,23.465,-43.044,-179.295,5.428,148.735
C09788=1222.574,23.714,-43.060,-179.293,5.427,148.734
C09789=1222.570,23.963,-43.075,-179.290,5.428,148.733
C09790=1222.564,24.213,-43.091,-179.288,5.428,148.733
C09791=1222.560,24.462,-43.106,-179.285,5.429,148.732
C09792=1222.555,24.712,-43.121,-179.282,5.429,148.731
C09793=1222.550,24.961,-43.136,-179.280,5.430,148.731
C09794=1222.545,25.210,-43.152,-179.278,5.430,148.730
C09795=1222.539,25.460,-43.167,-179.276,5.431,148.730
C09796=1222.534,25.709,-43.182,-179.273,5.431,148.729
C09797=1222.530,25.960,-43.198,-179.270,5.432,148.728
C09798=1222.524,26.209,-43.213,-179.268,5.432,148.728
C09799=1222.520,26.458,-43.228,-179.265,5.433,148.727
C09800=1222.514,26.707,-43.244,-179.262,5.433,148.726
C09801=1222.510,26.957,-43.259,-179.260,5.434,148.726
C09802=1222.505,27.207,-43.275,-179.258,5.434,148.725
C09803=1222.499,27.456,-43.291,-179.255,5.434,148.724
C09804=1222.495,27.705,-43.306,-179.252,5.435,148.723
C09805=1222.490,27.955,-43.322,-179.250,5.436,148.723
C09806=1222.484,28.205,-43.337,-179.247,5.436,148.722
C09807=1222.480,28.454,-43.352,-179.245,5.437,148.722
C09808=1222.474,28.703,-43.368,-179.242,5.437,148.721
C09809=1222.470,28.953,-43.384,-179.240,5.437,148.720
C09810=1222.464,29.222,-43.401,-179.237,5.438,148.720
C09811=1222.459,29.490,-43.417,-179.235,5.438,148.719
C09812=1222.454,29.758,-43.434,-179.232,5.439,148.718
C09813=1222.448,30.027,-43.450,-179.228,5.440,148.717
C09814=1222.443,30.277,-43.467,-179.226,5.439,148.717
C09815=1222.439,30.526,-43.482,-179.224,5.440,148.716
C09816=1222.433,30.775,-43.498,-179.222,5.441,148.716
C09817=1222.428,31.025,-43.513,-179.219,5.441,148.715
C09818=1222.423,31.275,-43.529,-179.216,5.442,148.714
C09819=1222.419,31.524,-43.544,-179.214,5.442,148.714
C09820=1222.413,31.773,-43.560,-179.211,5.443,148.713
C09821=1222.408,32.024,-43.576,-179.208,5.444,148.712
C09822=1222.403,32.272,-43.592,-179.206,5.443,148.711
C09823=1222.399,32.521,-43.607,-179.204,5.444,148.711
C09824=1222.394,32.772,-43.623,-179.201,5.444,148.710
C09825=1222.388,33.021,-43.639,-179.199,5.445,148.710
C09826=1222.383,33.270,-43.654,-179.196,5.446,148.709
C09827=1222.379,33.520,-43.670,-179.194,5.446,148.708
C09828=1222.374,33.769,-43.686,-179.191,5.447,148.708
C09829=1222.369,34.018,-43.701,-179.188,5.447,148.707
C09830=1222.364,34.268,-43.717,-179.186,5.448,148.706
C09831=1222.358,34.518,-43.733,-179.184,5.448,148.706
C09832=1222.354,34.766,-43.749,-179.181,5.448,148.705
C09833=1222.349,35.016,-43.765,-179.178,5.449,148.704
C09834=1222.344,35.266,-43.780,-179.176,5.450,148.704
C09835=1222.339,35.516,-43.796,-179.174,5.450,148.703
C09836=1222.334,35.765,-43.812,-179.171,5.451,148.702
C09837=1222.329,36.014,-43.828,-179.168,5.451,148.702
C09838=1222.324,36.264,-43.844,-179.166,5.452,148.701
C09839=1222.319,36.513,-43.859,-179.163,5.452,148.700
C09840=1222.314,36.762,-43.875,-179.160,5.453,148.700
C09841=1222.309,37.012,-43.891,-179.158,5.453,148.699
C09842=1222.304,37.262,-43.907,-179.156,5.453,148.698
C09843=1222.299,37.511,-43.923,-179.153,5.454,148.698
C09844=1222.294,37.760,-43.939,-179.151,5.455,148.697
C09845=1222.289,38.010,-43.955,-179.148,5.455,148.697
C09846=1222.284,38.259,-43.971,-179.146,5.456,148.696
C09847=1222.279,38.509,-43.987,-179.143,5.456,148.695
C09848=1222.275,38.759,-44.002,-179.140,5.457,148.695
C09849=1222.270,39.007,-44.019,-179.138,5.458,148.694
C09850=1222.264,39.257,-44.034,-179.135,5.458,148.693
C09851=1222.260,39.506,-44.051,-179.132,5.459,148.693
C09852=1222.254,39.756,-44.066,-179.130,5.460,148.692
C09853=1222.250,40.006,-44.082,-179.128,5.459,148.691
C09854=1222.245,40.255,-44.099,-179.125,5.460,148.691
C09855=1222.240,40.505,-44.115,-179.123,5.460,148.690
C09856=1222.235,40.753,-44.131,-179.120,5.461,148.689
C09857=1222.230,41.004,-44.147,-179.118,5.461,148.689
C09858=1222.225,41.252,-44.163,-179.115,5.462,148.688
C09859=1222.219,41.502,-44.179,-179.112,5.463,148.687
C09860=1222.215,41.751,-44.195,-179.110,5.464,148.687
C09861=1222.210,42.001,-44.211,-179.108,5.464,148.686
C09862=1222.205,42.251,-44.227,-179.105,5.465,148.686
C09863=1222.200,42.499,-44.243,-179.102,5.465,148.685
C09864=1222.195,42.750,-44.259,-179.100,5.466,148.684
C09865=1222.190,42.998,-44.276,-179.097,5.466,148.684
C09866=1222.185,43.248,-44.292,-179.094,5.467,148.683
C09867=1222.180,43.497,-44.308,-179.092,5.467,148.682
C09868=1222.175,43.747,-44.324,-179.090,5.467,148.682
C09869=1222.170,43.996,-44.340,-179.087,5.468,148.681
C09870=1222.166,44.246,-44.357,-179.085,5.469,148.680
C09871=1222.160,44.495,-44.372,-179.082,5.469,148.680
C09872=1222.156,44.744,-44.389,-179.080,5.470,148.679
C09873=1222.150,44.994,-44.405,-179.077,5.470,148.678
C09874=1222.146,45.243,-44.421,-179.074,5.471,148.678
C09875=1222.141,45.492,-44.438,-179.072,5.472,148.677
C09876=1222.135,45.743,-44.454,-179.069,5.472,148.677
C09877=1222.130,45.991,-44.470,-179.067,5.473,148.676
C09878=1222.125,46.241,-44.486,-179.064,5.473,148.675
C09879=1222.120,46.490,-44.503,-179.062,5.474,148.675
C09880=1222.116,46.740,-44.519,-179.059,5.475,148.674
C09881=1222.111,46.990,-44.535,-179.056,5.475,148.673
C09882=1222.106,47.239,-44.552,-179.054,5.476,148.673
C09883=1222.102,47.488,-44.568,-179.052,5.477,148.672
C09884=1222.096,47.738,-44.584,-179.049,5.477,148.672
C09885=1222.092,47.987,-44.601,-179.046,5.478,148.671
C09886=1222.086,48.236,-44.617,-179.044,5.477,148.670
C09887=1222.081,48.486,-44.633,-179.042,5.478,148.670
C09888=1222.076,48.735,-44.650,-179.039,5.479,148.669
C09889=1222.071,48.984,-44.666,-179.037,5.479,148.668
C09890=1222.067,49.235,-44.682,-179.034,5.480,148.668
C09891=1222.062,49.483,-44.699,-179.031,5.481,148.667
C09892=1222.056,49.733,-44.716,-179.029,5.481,148.666
C09893=1222.051,49.982,-44.732,-179.026,5.482,148.666
C09894=1222.047,50.232,-44.748,-179.024,5.482,148.665
C09895=1222.042,50.482,-44.765,-179.021,5.483,148.664
C09896=1222.037,50.730,-44.781,-179.019,5.484,148.664
C09897=1222.032,50.980,-44.798,-179.016,5.484,148.663
C09898=1222.026,51.229,-44.814,-179.014,5.485,148.663
C09899=1222.022,51.479,-44.831,-179.011,5.485,148.662
C09900=1222.017,51.728,-44.847,-179.008,5.486,148.661
C09901=1222.012,51.977,-44.864,-179.006,5.487,148.661
C09902=1222.007,52.227,-44.881,-179.003,5.487,148.660
C09903=1222.003,52.477,-44.898,-179.001,5.488,148.660
C09904=1221.997,52.726,-44.913,-178.998,5.489,148.659
C09905=1221.993,52.975,-44.930,-178.996,5.489,148.658
C09906=1221.988,53.224,-44.946,-178.993,5.490,148.657
C09907=1221.982,53.474,-44.963,-178.990,5.490,148.657
C09908=1221.978,53.723,-44.980,-178.988,5.491,148.656
C09909=1221.973,53.972,-44.996,-178.985,5.492,148.656
C09910=1221.968,54.222,-45.014,-178.983,5.492,148.655
C09911=1221.963,54.472,-45.030,-178.980,5.493,148.654
C09912=1221.958,54.721,-45.046,-178.978,5.493,148.654
C09913=1221.953,54.970,-45.063,-178.975,5.494,148.653
C09914=1221.947,55.239,-45.081,-178.972,5.495,148.652
C09915=1221.943,55.507,-45.099,-178.970,5.495,148.652
C09916=1221.937,55.775,-45.117,-178.967,5.496,148.651
C09917=1221.932,56.045,-45.135,-178.964,5.496,148.650
C09918=1221.927,56.294,-45.151,-178.962,5.497,148.650
C09919=1221.921,56.543,-45.168,-178.960,5.498,148.649
C09920=1221.917,56.793,-45.185,-178.957,5.498,148.649
C09921=1221.912,57.042,-45.202,-178.954,5.499,148.648
C09922=1221.907,57.291,-45.218,-178.952,5.499,148.647
C09923=1221.902,57.541,-45.235,-178.949,5.500,148.647
C09924=1221.898,57.790,-45.252,-178.946,5.501,148.646
C09925=1221.892,58.039,-45.269,-178.944,5.502,148.646
C09926=1221.887,58.289,-45.285,-178.942,5.502,148.645
C09927=1221.883,58.538,-45.302,-178.939,5.503,148.644
C09928=1221.878,58.788,-45.319,-178.936,5.503,148.644
C09929=1221.873,59.037,-45.336,-178.934,5.504,148.643
C09930=1221.867,59.287,-45.353,-178.932,5.505,148.642
C09931=1221.863,59.535,-45.370,-178.929,5.505,148.642
C09932=1221.859,59.785,-45.387,-178.926,5.506,148.641
C09933=1221.853,60.034,-45.404,-178.924,5.506,148.640
C09934=1221.848,60.283,-45.420,-178.921,5.507,148.640
C09935=1221.843,60.533,-45.438,-178.919,5.508,148.639
C09936=1221.839,60.783,-45.454,-178.916,5.509,148.639
C09937=1221.833,61.032,-45.471,-178.913,5.510,148.638
C09938=1221.828,61.281,-45.488,-178.910,5.510,148.637
C09939=1221.823,61.531,-45.505,-178.908,5.511,148.637
C09940=1221.819,61.780,-45.523,-178.905,5.512,148.636
C09941=1221.814,62.029,-45.539,-178.903,5.513,148.636
C09942=1221.809,62.279,-45.556,-178.900,5.513,148.635
C09943=1221.804,62.528,-45.573,-178.898,5.514,148.634
C09944=1221.799,62.778,-45.590,-178.895,5.514,148.634
C09945=1221.794,63.027,-45.606,-178.893,5.515,148.633
C09946=1221.789,63.276,-45.624,-178.890,5.516,148.632
C09947=1221.785,63.525,-45.641,-178.888,5.516,148.632
C09948=1221.779,63.775,-45.658,-178.885,5.517,148.631
C09949=1221.775,64.025,-45.675,-178.883,5.517,148.630
C09950=1221.770,64.274,-45.692,-178.880,5.518,148.630
C09951=1221.765,64.523,-45.709,-178.878,5.519,148.629
C09952=1221.760,64.772,-45.727,-178.875,5.520,148.629
C09953=1221.755,65.022,-45.743,-178.872,5.520,148.628
C09954=1221.750,65.272,-45.761,-178.870,5.521,148.627
C09955=1221.745,65.521,-45.778,-178.868,5.522,148.627
C09956=1221.740,65.770,-45.795,-178.865,5.522,148.626
C09957=1221.735,66.019,-45.812,-178.862,5.523,148.626
C09958=1221.731,66.268,-45.829,-178.860,5.523,148.625
C09959=1221.725,66.518,-45.847,-178.857,5.524,148.624
C09960=1221.721,66.768,-45.863,-178.855,5.525,148.624
C09961=1221.716,67.017,-45.881,-178.852,5.525,148.623
C09962=1221.711,67.266,-45.899,-178.850,5.526,148.623
C09963=1221.706,67.515,-45.915,-178.847,5.527,148.622
C09964=1221.701,67.764,-45.933,-178.845,5.527,148.621
C09965=1221.696,68.014,-45.950,-178.842,5.529,148.621
C09966=1221.691,68.264,-45.967,-178.839,5.529,148.620
C09967=1221.686,68.513,-45.985,-178.837,5.530,148.619
C09968=1221.682,68.762,-46.001,-178.834,5.531,148.619
C09969=1221.676,69.012,-46.019,-178.832,5.532,148.618
C09970=1221.672,69.261,-46.036,-178.829,5.532,148.618
C09971=1221.666,69.510,-46.053,-178.827,5.533,148.617
C09972=1221.662,69.759,-46.071,-178.824,5.533,148.616
C09973=1221.657,70.009,-46.088,-178.821,5.534,148.616
C09974=1221.652,70.258,-46.106,-178.819,5.535,148.615
C09975=1221.647,70.508,-46.123,-178.817,5.535,148.615
C09976=1221.642,70.757,-46.140,-178.814,5.536,148.614
C09977=1221.638,71.006,-46.158,-178.811,5.537,148.613
C09978=1221.632,71.256,-46.175,-178.809,5.537,148.613
C09979=1221.628,71.505,-46.192,-178.806,5.538,148.612
C09980=1221.623,71.755,-46.209,-178.803,5.539,148.612
C09981=1221.618,72.004,-46.227,-178.801,5.540,148.611
C09982=1221.613,72.253,-46.244,-178.799,5.541,148.610
C09983=1221.608,72.502,-46.262,-178.796,5.542,148.610
C09984=1221.603,72.752,-46.279,-178.793,5.542,148.609
C09985=1221.598,73.001,-46.297,-178.791,5.543,148.609
C09986=1221.593,73.250,-46.314,-178.789,5.544,148.608
C09987=1221.589,73.500,-46.332,-178.786,5.544,148.607
C09988=1221.584,73.749,-46.350,-178.783,5.545,148.607
C09989=1221.578,73.999,-46.367,-178.781,5.545,148.606
C09990=1221.574,74.247,-46.384,-178.778,5.546,148.605
C09991=1221.569,74.497,-46.402,-178.776,5.547,148.605
C09992=1221.564,74.746,-46.420,-178.773,5.547,148.604
C09993=1221.559,74.996,-46.437,-178.770,5.549,148.604
C09994=1221.555,75.245,-46.454,-178.767,5.549,148.603
C09995=1221.550,75.494,-46.472,-178.765,5.550,148.603
C09996=1221.545,75.744,-46.489,-178.763,5.551,148.602
//INST
///DATE 2021/06/15 17:22
///ATTR SC,RW,RJ
////FRAME ROBOT
///GROUP1 RB1
NOP
MOVL C00000 V=800.0 PL=0
MOVL C00001 V=800.0 PL=0
MOVL C00002 V=800.0 PL=0
MOVL C00003 V=800.0 PL=0
MOVL C00004 V=800.0 PL=0
MOVL C00005 V=800.0 PL=0
MOVL C00006 V=800.0 PL=0
MOVL C00007 V=800.0 PL=0
MOVL C00008 V=800.0 PL=0
MOVL C00009 V=800.0 PL=0
MOVL C00010 V=800.0 PL=0
MOVL C00011 V=800.0 PL=0
MOVL C00012 V=800.0 PL=0
MOVL C00013 V=800.0 PL=0
MOVL C00014 V=800.0 PL=0
MOVL C00015 V=800.0 PL=0
MOVL C00016 V=800.0 PL=0
MOVL C00017 V=800.0 PL=0
MOVL C00018 V=800.0 PL=0
MOVL C00019 V=800.0 PL=0
MOVL C00020 V=800.0 PL=0
MOVL C00021 V=800.0 PL=0
MOVL C00022 V=800.0 PL=0
MOVL C00023 V=800.0 PL=0
MOVL C00024 V=800.0 PL=0
MOVL C00025 V=800.0 PL=0
MOVL C00026 V=800.0 PL=0
MOVL C00027 V=800.0 PL=0
MOVL C00028 V=800.0 PL=0
MOVL C00029 V=800.0 PL=0
MOVL C00030 V=800.0 PL=0
MOVL C00031 V=800.0 PL=0
MOVL C00032 V=800.0 PL=0
MOVL C00033 V=800.0 PL=0
MOVL C00034 V=800.0 PL=0
MOVL C00035 V=800.0 PL=0
MOVL C00036 V=800.0 PL=0
MOVL C00037 V=800.0 PL=0
MOVL C00038 V=800.0 PL=0
MOVL C00039 V=800.0 PL=0
MOVL C00040 V=800.0 PL=0
MOVL C00041 V=800.0 PL=0
MOVL C00042 V=800.0 PL=0
MOVL C00043 V=800.0 PL=0
MOVL C00044 V=800.0 PL=0
MOVL C00045 V=800.0 PL=0
MOVL C00046 V=800.0 PL=0
MOVL C00047 V=800.0 PL=0
MOVL C00048 V=800.0 PL=0
MOVL C00049 V=800.0 PL=0
MOVL C00050 V=800.0 PL=0
MOVL C00051 V=800.0 PL=0
MOVL C00052 V=800.0 PL=0
MOVL C00053 V=800.0 PL=0
MOVL C00054 V=800.0 PL=0
MOVL C00055 V=800.0 PL=0
MOVL C00056 V=800.0 PL=0
MOVL C00057 V=800.0 PL=0
MOVL C00058 V=800.0 PL=0
MOVL C00059 V=800.0 PL=0
MOVL C00060 V=800.0 PL=0
MOVL C00061 V=800.0 PL=0
MOVL C00062 V=800.0 PL=0
MOVL C00063 V=800.0 PL=0
MOVL C00064 V=800.0 PL=0
MOVL C00065 V=800.0 PL=0
MOVL C00066 V=800.0 PL=0
MOVL C00067 V=800.0 PL=0
MOVL C00068 V=800.0 PL=0
MOVL C00069 V=800.0 PL=0
MOVL C00070 V=800.0 PL=0
MOVL C00071 V=800.0 PL=0
MOVL C00072 V=800.0 PL=0
MOVL C00073 V=800.0 PL=0
MOVL C00074 V=800.0 PL=0
MOVL C00075 V=800.0 PL=0
MOVL C00076 V=800.0 PL=0
MOVL C00077 V=800.0 PL=0
MOVL C00078 V=800.0 PL=0
MOVL C00079 V=800.0 PL=0
MOVL C00080 V=800.0 PL=0
MOVL C00081 V=800.0 PL=0
MOVL C00082 V=800.0 PL=0
MOVL C00083 V=800.0 PL=0
MOVL C00084 V=800.0 PL=0
MOVL C00085 V=800.0 PL=0
MOVL C00086 V=800.0 PL=0
MOVL C00087 V=800.0 PL=0
MOVL C00088 V=800.0 PL=0
MOVL C00089 V=800.0 PL=0
MOVL C00090 V=800.0 PL=0
MOVL C00091 V=800.0 PL=0
MOVL C00092 V=800.0 PL=0
MOVL C00093 V=800.0 PL=0
MOVL C00094 V=800.0 PL=0
MOVL C00095 V=800.0 PL=0
MOVL C00096 V=800.0 PL=0
MOVL C00097 V=800.0 PL=0
MOVL C00098 V=800.0 PL=0
MOVL C00099 V=800.0 PL=0
MOVL C00100 V=800.0 PL=0
MOVL C00101 V=800.0 PL=0
MOVL C00102 V=800.0 PL=0
MOVL C00103 V=800.0 PL=0
MOVL C00104 V=800.0 PL=0
MOVL C00105 V=800.0 PL=0
MOVL C00106 V=800.0 PL=0
MOVL C00107 V=800.0 PL=0
MOVL C00108 V=800.0 PL=0
MOVL C00109 V=800.0 PL=0
MOVL C00110 V=800.0 PL=0
MOVL C00111 V=800.0 PL=0
MOVL C00112 V=800.0 PL=0
MOVL C00113 V=800.0 PL=0
MOVL C00114 V=800.0 PL=0
MOVL C00115 V=800.0 PL=0
MOVL C00116 V=800.0 PL=0
MOVL C00117 V=800.0 PL=0
MOVL C00118 V=800.0 PL=0
MOVL C00119 V=800.0 PL=0
MOVL C00120 V=800.0 PL=0
MOVL C00121 V=800.0 PL=0
MOVL C00122 V=800.0 PL=0
MOVL C00123 V=800.0 PL=0
MOVL C00124 V=800.0 PL=0
MOVL C00125 V=800.0 PL=0
MOVL C00126 V=800.0 PL=0
MOVL C00127 V=800.0 PL=0
MOVL C00128 V=800.0 PL=0
MOVL C00129 V=800.0 PL=0
MOVL C00130 V=800.0 PL=0
MOVL C00131 V=800.0 PL=0
MOVL C00132 V=800.0 PL=0
MOVL C00133 V=800.0 PL=0
MOVL C00134 V=800.0 PL=0
MOVL C00135 V=800.0 PL=0
MOVL C00136 V=800.0 PL=0
MOVL C00137 V=800.0 PL=0
MOVL C00138 V=800.0 PL=0
MOVL C00139 V=800.0 PL=0
MOVL C00140 V=800.0 PL=0
MOVL C00141 V=800.0 PL=0
MOVL C00142 V=800.0 PL=0
MOVL C00143 V=800.0 PL=0
MOVL C00144 V=800.0 PL=0
MOVL C00145 V=800.0 PL=0
MOVL C00146 V=800.0 PL=0
MOVL C00147 V=800.0 PL=0
MOVL C00148 V=800.0 PL=0
MOVL C00149 V=800.0 PL=0
MOVL C00150 V=800.0 PL=0
MOVL C00151 V=800.0 PL=0
MOVL C00152 V=800.0 PL=0
MOVL C00153 V=800.0 PL=0
MOVL C00154 V=800.0 PL=0
MOVL C00155 V=800.0 PL=0
MOVL C00156 V=800.0 PL=0
MOVL C00157 V=800.0 PL=0
MOVL C00158 V=800.0 PL=0
MOVL C00159 V=800.0 PL=0
MOVL C00160 V=800.0 PL=0
MOVL C00161 V=800.0 PL=0
MOVL C00162 V=800.0 PL=0
MOVL C00163 V=800.0 PL=0
MOVL C00164 V=800.0 PL=0
MOVL C00165 V=800.0 PL=0
MOVL C00166 V=800.0 PL=0
MOVL C00167 V=800.0 PL=0
MOVL C00168 V=800.0 PL=0
MOVL C00169 V=800.0 PL=0
MOVL C00170 V=800.0 PL=0
MOVL C00171 V=800.0 PL=0
MOVL C00172 V=800.0 PL=0
MOVL C00173 V=800.0 PL=0
MOVL C00174 V=800.0 PL=0
MOVL C00175 V=800.0 PL=0
MOVL C00176 V=800.0 PL=0
MOVL C00177 V=800.0 PL=0
MOVL C00178 V=800.0 PL=0
MOVL C00179 V=800.0 PL=0
MOVL C00180 V=800.0 PL=0
MOVL C00181 V=800.0 PL=0
MOVL C00182 V=800.0 PL=0
MOVL C00183 V=800.0 PL=0
MOVL C00184 V=800.0 PL=0
MOVL C00185 V=800.0 PL=0
MOVL C00186 V=800.0 PL=0
MOVL C00187 V=800.0 PL=0
MOVL C00188 V=800.0 PL=0
MOVL C00189 V=800.0 PL=0
MOVL C00190 V=800.0 PL=0
MOVL C00191 V=800.0 PL=0
MOVL C00192 V=800.0 PL=0
MOVL C00193 V=800.0 PL=0
MOVL C00194 V=800.0 PL=0
MOVL C00195 V=800.0 PL=0
MOVL C00196 V=800.0 PL=0
MOVL C00197 V=800.0 PL=0
MOVL C00198 V=800.0 PL=0
MOVL C00199 V=800.0 PL=0
MOVL C00200 V=800.0 PL=0
MOVL C00201 V=800.0 PL=0
MOVL C00202 V=800.0 PL=0
MOVL C00203 V=800.0 PL=0
MOVL C00204 V=800.0 PL=0
MOVL C00205 V=800.0 PL=0
MOVL C00206 V=800.0 PL=0
MOVL C00207 V=800.0 PL=0
MOVL C00208 V=800.0 PL=0
MOVL C00209 V=800.0 PL=0
MOVL C00210 V=800.0 PL=0
MOVL C00211 V=800.0 PL=0
MOVL C00212 V=800.0 PL=0
MOVL C00213 V=800.0 PL=0
MOVL C00214 V=800.0 PL=0
MOVL C00215 V=800.0 PL=0
MOVL C00216 V=800.0 PL=0
MOVL C00217 V=800.0 PL=0
MOVL C00218 V=800.0 PL=0
MOVL C00219 V=800.0 PL=0
MOVL C00220 V=800.0 PL=0
MOVL C00221 V=800.0 PL=0
MOVL C00222 V=800.0 PL=0
MOVL C00223 V=800.0 PL=0
MOVL C00224 V=800.0 PL=0
MOVL C00225 V=800.0 PL=0
MOVL C00226 V=800.0 PL=0
MOVL C00227 V=800.0 PL=0
MOVL C00228 V=800.0 PL=0
MOVL C00229 V=800.0 PL=0
MOVL C00230 V=800.0 PL=0
MOVL C00231 V=800.0 PL=0
MOVL C00232 V=800.0 PL=0
MOVL C00233 V=800.0 PL=0
MOVL C00234 V=800.0 PL=0
MOVL C00235 V=800.0 PL=0
MOVL C00236 V=800.0 PL=0
MOVL C00237 V=800.0 PL=0
MOVL C00238 V=800.0 PL=0
MOVL C00239 V=800.0 PL=0
MOVL C00240 V=800.0 PL=0
MOVL C00241 V=800.0 PL=0
MOVL C00242 V=800.0 PL=0
MOVL C00243 V=800.0 PL=0
MOVL C00244 V=800.0 PL=0
MOVL C00245 V=800.0 PL=0
MOVL C00246 V=800.0 PL=0
MOVL C00247 V=800.0 PL=0
MOVL C00248 V=800.0 PL=0
MOVL C00249 V=800.0 PL=0
MOVL C00250 V=800.0 PL=0
MOVL C00251 V=800.0 PL=0
MOVL C00252 V=800.0 PL=0
MOVL C00253 V=800.0 PL=0
MOVL C00254 V=800.0 PL=0
MOVL C00255 V=800.0 PL=0
MOVL C00256 V=800.0 PL=0
MOVL C00257 V=800.0 PL=0
MOVL C00258 V=800.0 PL=0
MOVL C00259 V=800.0 PL=0
MOVL C00260 V=800.0 PL=0
MOVL C00261 V=800.0 PL=0
MOVL C00262 V=800.0 PL=0
MOVL C00263 V=800.0 PL=0
MOVL C00264 V=800.0 PL=0
MOVL C00265 V=800.0 PL=0
MOVL C00266 V=800.0 PL=0
MOVL C00267 V=800.0 PL=0
MOVL C00268 V=800.0 PL=0
MOVL C00269 V=800.0 PL=0
MOVL C00270 V=800.0 PL=0
MOVL C00271 V=800.0 PL=0
MOVL C00272 V=800.0 PL=0
MOVL C00273 V=800.0 PL=0
MOVL C00274 V=800.0 PL=0
MOVL C00275 V=800.0 PL=0
MOVL C00276 V=800.0 PL=0
MOVL C00277 V=800.0 PL=0
MOVL C00278 V=800.0 PL=0
MOVL C00279 V=800.0 PL=0
MOVL C00280 V=800.0 PL=0
MOVL C00281 V=800.0 PL=0
MOVL C00282 V=800.0 PL=0
MOVL C00283 V=800.0 PL=0
MOVL C00284 V=800.0 PL=0
MOVL C00285 V=800.0 PL=0
MOVL C00286 V=800.0 PL=0
MOVL C00287 V=800.0 PL=0
MOVL C00288 V=800.0 PL=0
MOVL C00289 V=800.0 PL=0
MOVL C00290 V=800.0 PL=0
MOVL C00291 V=800.0 PL=0
MOVL C00292 V=800.0 PL=0
MOVL C00293 V=800.0 PL=0
MOVL C00294 V=800.0 PL=0
MOVL C00295 V=800.0 PL=0
MOVL C00296 V=800.0 PL=0
MOVL C00297 V=800.0 PL=0
MOVL C00298 V=800.0 PL=0
MOVL C00299 V=800.0 PL=0
MOVL C00300 V=800.0 PL=0
MOVL C00301 V=800.0 PL=0
MOVL C00302 V=800.0 PL=0
MOVL C00303 V=800.0 PL=0
MOVL C00304 V=800.0 PL=0
MOVL C00305 V=800.0 PL=0
MOVL C00306 V=800.0 PL=0
MOVL C00307 V=800.0 PL=0
MOVL C00308 V=800.0 PL=0
MOVL C00309 V=800.0 PL=0
MOVL C00310 V=800.0 PL=0
MOVL C00311 V=800.0 PL=0
MOVL C00312 V=800.0 PL=0
MOVL C00313 V=800.0 PL=0
MOVL C00314 V=800.0 PL=0
MOVL C00315 V=800.0 PL=0
MOVL C00316 V=800.0 PL=0
MOVL C00317 V=800.0 PL=0
MOVL C00318 V=800.0 PL=0
MOVL C00319 V=800.0 PL=0
MOVL C00320 V=800.0 PL=0
MOVL C00321 V=800.0 PL=0
MOVL C00322 V=800.0 PL=0
MOVL C00323 V=800.0 PL=0
MOVL C00324 V=800.0 PL=0
MOVL C00325 V=800.0 PL=0
MOVL C00326 V=800.0 PL=0
MOVL C00327 V=800.0 PL=0
MOVL C00328 V=800.0 PL=0
MOVL C00329 V=800.0 PL=0
MOVL C00330 V=800.0 PL=0
MOVL C00331 V=800.0 PL=0
MOVL C00332 V=800.0 PL=0
MOVL C00333 V=800.0 PL=0
MOVL C00334 V=800.0 PL=0
MOVL C00335 V=800.0 PL=0
MOVL C00336 V=800.0 PL=0
MOVL C00337 V=800.0 PL=0
MOVL C00338 V=800.0 PL=0
MOVL C00339 V=800.0 PL=0
MOVL C00340 V=800.0 PL=0
MOVL C00341 V=800.0 PL=0
MOVL C00342 V=800.0 PL=0
MOVL C00343 V=800.0 PL=0
MOVL C00344 V=800.0 PL=0
MOVL C00345 V=800.0 PL=0
MOVL C00346 V=800.0 PL=0
MOVL C00347 V=800.0 PL=0
MOVL C00348 V=800.0 PL=0
MOVL C00349 V=800.0 PL=0
MOVL C00350 V=800.0 PL=0
MOVL C00351 V=800.0 PL=0
MOVL C00352 V=800.0 PL=0
MOVL C00353 V=800.0 PL=0
MOVL C00354 V=800.0 PL=0
MOVL C00355 V=800.0 PL=0
MOVL C00356 V=800.0 PL=0
MOVL C00357 V=800.0 PL=0
MOVL C00358 V=800.0 PL=0
MOVL C00359 V=800.0 PL=0
MOVL C00360 V=800.0 PL=0
MOVL C00361 V=800.0 PL=0
MOVL C00362 V=800.0 PL=0
MOVL C00363 V=800.0 PL=0
MOVL C00364 V=800.0 PL=0
MOVL C00365 V=800.0 PL=0
MOVL C00366 V=800.0 PL=0
MOVL C00367 V=800.0 PL=0
MOVL C00368 V=800.0 PL=0
MOVL C00369 V=800.0 PL=0
MOVL C00370 V=800.0 PL=0
MOVL C00371 V=800.0 PL=0
MOVL C00372 V=800.0 PL=0
MOVL C00373 V=800.0 PL=0
MOVL C00374 V=800.0 PL=0
MOVL C00375 V=800.0 PL=0
MOVL C00376 V=800.0 PL=0
MOVL C00377 V=800.0 PL=0
MOVL C00378 V=800.0 PL=0
MOVL C00379 V=800.0 PL=0
MOVL C00380 V=800.0 PL=0
MOVL C00381 V=800.0 PL=0
MOVL C00382 V=800.0 PL=0
MOVL C00383 V=800.0 PL=0
MOVL C00384 V=800.0 PL=0
MOVL C00385 V=800.0 PL=0
MOVL C00386 V=800.0 PL=0
MOVL C00387 V=800.0 PL=0
MOVL C00388 V=800.0 PL=0
MOVL C00389 V=800.0 PL=0
MOVL C00390 V=800.0 PL=0
MOVL C00391 V=800.0 PL=0
MOVL C00392 V=800.0 PL=0
MOVL C00393 V=800.0 PL=0
MOVL C00394 V=800.0 PL=0
MOVL C00395 V=800.0 PL=0
MOVL C00396 V=800.0 PL=0
MOVL C00397 V=800.0 PL=0
MOVL C00398 V=800.0 PL=0
MOVL C00399 V=800.0 PL=0
MOVL C00400 V=800.0 PL=0
MOVL C00401 V=800.0 PL=0
MOVL C00402 V=800.0 PL=0
MOVL C00403 V=800.0 PL=0
MOVL C00404 V=800.0 PL=0
MOVL C00405 V=800.0 PL=0
MOVL C00406 V=800.0 PL=0
MOVL C00407 V=800.0 PL=0
MOVL C00408 V=800.0 PL=0
MOVL C00409 V=800.0 PL=0
MOVL C00410 V=800.0 PL=0
MOVL C00411 V=800.0 PL=0
MOVL C00412 V=800.0 PL=0
MOVL C00413 V=800.0 PL=0
MOVL C00414 V=800.0 PL=0
MOVL C00415 V=800.0 PL=0
MOVL C00416 V=800.0 PL=0
MOVL C00417 V=800.0 PL=0
MOVL C00418 V=800.0 PL=0
MOVL C00419 V=800.0 PL=0
MOVL C00420 V=800.0 PL=0
MOVL C00421 V=800.0 PL=0
MOVL C00422 V=800.0 PL=0
MOVL C00423 V=800.0 PL=0
MOVL C00424 V=800.0 PL=0
MOVL C00425 V=800.0 PL=0
MOVL C00426 V=800.0 PL=0
MOVL C00427 V=800.0 PL=0
MOVL C00428 V=800.0 PL=0
MOVL C00429 V=800.0 PL=0
MOVL C00430 V=800.0 PL=0
MOVL C00431 V=800.0 PL=0
MOVL C00432 V=800.0 PL=0
MOVL C00433 V=800.0 PL=0
MOVL C00434 V=800.0 PL=0
MOVL C00435 V=800.0 PL=0
MOVL C00436 V=800.0 PL=0
MOVL C00437 V=800.0 PL=0
MOVL C00438 V=800.0 PL=0
MOVL C00439 V=800.0 PL=0
MOVL C00440 V=800.0 PL=0
MOVL C00441 V=800.0 PL=0
MOVL C00442 V=800.0 PL=0
MOVL C00443 V=800.0 PL=0
MOVL C00444 V=800.0 PL=0
MOVL C00445 V=800.0 PL=0
MOVL C00446 V=800.0 PL=0
MOVL C00447 V=800.0 PL=0
MOVL C00448 V=800.0 PL=0
MOVL C00449 V=800.0 PL=0
MOVL C00450 V=800.0 PL=0
MOVL C00451 V=800.0 PL=0
MOVL C00452 V=800.0 PL=0
MOVL C00453 V=800.0 PL=0
MOVL C00454 V=800.0 PL=0
MOVL C00455 V=800.0 PL=0
MOVL C00456 V=800.0 PL=0
MOVL C00457 V=800.0 PL=0
MOVL C00458 V=800.0 PL=0
MOVL C00459 V=800.0 PL=0
MOVL C00460 V=800.0 PL=0
MOVL C00461 V=800.0 PL=0
MOVL C00462 V=800.0 PL=0
MOVL C00463 V=800.0 PL=0
MOVL C00464 V=800.0 PL=0
MOVL C00465 V=800.0 PL=0
MOVL C00466 V=800.0 PL=0
MOVL C00467 V=800.0 PL=0
MOVL C00468 V=800.0 PL=0
MOVL C00469 V=800.0 PL=0
MOVL C00470 V=800.0 PL=0
MOVL C00471 V=800.0 PL=0
MOVL C00472 V=800.0 PL=0
MOVL C00473 V=800.0 PL=0
MOVL C00474 V=800.0 PL=0
MOVL C00475 V=800.0 PL=0
MOVL C00476 V=800.0 PL=0
MOVL C00477 V=800.0 PL=0
MOVL C00478 V=800.0 PL=0
MOVL C00479 V=800.0 PL=0
MOVL C00480 V=800.0 PL=0
MOVL C00481 V=800.0 PL=0
MOVL C00482 V=800.0 PL=0
MOVL C00483 V=800.0 PL=0
MOVL C00484 V=800.0 PL=0
MOVL C00485 V=800.0 PL=0
MOVL C00486 V=800.0 PL=0
MOVL C00487 V=800.0 PL=0
MOVL C00488 V=800.0 PL=0
MOVL C00489 V=800.0 PL=0
MOVL C00490 V=800.0 PL=0
MOVL C00491 V=800.0 PL=0
MOVL C00492 V=800.0 PL=0
MOVL C00493 V=800.0 PL=0
MOVL C00494 V=800.0 PL=0
MOVL C00495 V=800.0 PL=0
MOVL C00496 V=800.0 PL=0
MOVL C00497 V=800.0 PL=0
MOVL C00498 V=800.0 PL=0
MOVL C00499 V=800.0 PL=0
MOVL C00500 V=800.0 PL=0
MOVL C00501 V=800.0 PL=0
MOVL C00502 V=800.0 PL=0
MOVL C00503 V=800.0 PL=0
MOVL C00504 V=800.0 PL=0
MOVL C00505 V=800.0 PL=0
MOVL C00506 V=800.0 PL=0
MOVL C00507 V=800.0 PL=0
MOVL C00508 V=800.0 PL=0
MOVL C00509 V=800.0 PL=0
MOVL C00510 V=800.0 PL=0
MOVL C00511 V=800.0 PL=0
MOVL C00512 V=800.0 PL=0
MOVL C00513 V=800.0 PL=0
MOVL C00514 V=800.0 PL=0
MOVL C00515 V=800.0 PL=0
MOVL C00516 V=800.0 PL=0
MOVL C00517 V=800.0 PL=0
MOVL C00518 V=800.0 PL=0
MOVL C00519 V=800.0 PL=0
MOVL C00520 V=800.0 PL=0
MOVL C00521 V=800.0 PL=0
MOVL C00522 V=800.0 PL=0
MOVL C00523 V=800.0 PL=0
MOVL C00524 V=800.0 PL=0
MOVL C00525 V=800.0 PL=0
MOVL C00526 V=800.0 PL=0
MOVL C00527 V=800.0 PL=0
MOVL C00528 V=800.0 PL=0
MOVL C00529 V=800.0 PL=0
MOVL C00530 V=800.0 PL=0
MOVL C00531 V=800.0 PL=0
MOVL C00532 V=800.0 PL=0
MOVL C00533 V=800.0 PL=0
MOVL C00534 V=800.0 PL=0
MOVL C00535 V=800.0 PL=0
MOVL C00536 V=800.0 PL=0
MOVL C00537 V=800.0 PL=0
MOVL C00538 V=800.0 PL=0
MOVL C00539 V=800.0 PL=0
MOVL C00540 V=800.0 PL=0
MOVL C00541 V=800.0 PL=0
MOVL C00542 V=800.0 PL=0
MOVL C00543 V=800.0 PL=0
MOVL C00544 V=800.0 PL=0
MOVL C00545 V=800.0 PL=0
MOVL C00546 V=800.0 PL=0
MOVL C00547 V=800.0 PL=0
MOVL C00548 V=800.0 PL=0
MOVL C00549 V=800.0 PL=0
MOVL C00550 V=800.0 PL=0
MOVL C00551 V=800.0 PL=0
MOVL C00552 V=800.0 PL=0
MOVL C00553 V=800.0 PL=0
MOVL C00554 V=800.0 PL=0
MOVL C00555 V=800.0 PL=0
MOVL C00556 V=800.0 PL=0
MOVL C00557 V=800.0 PL=0
MOVL C00558 V=800.0 PL=0
MOVL C00559 V=800.0 PL=0
MOVL C00560 V=800.0 PL=0
MOVL C00561 V=800.0 PL=0
MOVL C00562 V=800.0 PL=0
MOVL C00563 V=800.0 PL=0
MOVL C00564 V=800.0 PL=0
MOVL C00565 V=800.0 PL=0
MOVL C00566 V=800.0 PL=0
MOVL C00567 V=800.0 PL=0
MOVL C00568 V=800.0 PL=0
MOVL C00569 V=800.0 PL=0
MOVL C00570 V=800.0 PL=0
MOVL C00571 V=800.0 PL=0
MOVL C00572 V=800.0 PL=0
MOVL C00573 V=800.0 PL=0
MOVL C00574 V=800.0 PL=0
MOVL C00575 V=800.0 PL=0
MOVL C00576 V=800.0 PL=0
MOVL C00577 V=800.0 PL=0
MOVL C00578 V=800.0 PL=0
MOVL C00579 V=800.0 PL=0
MOVL C00580 V=800.0 PL=0
MOVL C00581 V=800.0 PL=0
MOVL C00582 V=800.0 PL=0
MOVL C00583 V=800.0 PL=0
MOVL C00584 V=800.0 PL=0
MOVL C00585 V=800.0 PL=0
MOVL C00586 V=800.0 PL=0
MOVL C00587 V=800.0 PL=0
MOVL C00588 V=800.0 PL=0
MOVL C00589 V=800.0 PL=0
MOVL C00590 V=800.0 PL=0
MOVL C00591 V=800.0 PL=0
MOVL C00592 V=800.0 PL=0
MOVL C00593 V=800.0 PL=0
MOVL C00594 V=800.0 PL=0
MOVL C00595 V=800.0 PL=0
MOVL C00596 V=800.0 PL=0
MOVL C00597 V=800.0 PL=0
MOVL C00598 V=800.0 PL=0
MOVL C00599 V=800.0 PL=0
MOVL C00600 V=800.0 PL=0
MOVL C00601 V=800.0 PL=0
MOVL C00602 V=800.0 PL=0
MOVL C00603 V=800.0 PL=0
MOVL C00604 V=800.0 PL=0
MOVL C00605 V=800.0 PL=0
MOVL C00606 V=800.0 PL=0
MOVL C00607 V=800.0 PL=0
MOVL C00608 V=800.0 PL=0
MOVL C00609 V=800.0 PL=0
MOVL C00610 V=800.0 PL=0
MOVL C00611 V=800.0 PL=0
MOVL C00612 V=800.0 PL=0
MOVL C00613 V=800.0 PL=0
MOVL C00614 V=800.0 PL=0
MOVL C00615 V=800.0 PL=0
MOVL C00616 V=800.0 PL=0
MOVL C00617 V=800.0 PL=0
MOVL C00618 V=800.0 PL=0
MOVL C00619 V=800.0 PL=0
MOVL C00620 V=800.0 PL=0
MOVL C00621 V=800.0 PL=0
MOVL C00622 V=800.0 PL=0
MOVL C00623 V=800.0 PL=0
MOVL C00624 V=800.0 PL=0
MOVL C00625 V=800.0 PL=0
MOVL C00626 V=800.0 PL=0
MOVL C00627 V=800.0 PL=0
MOVL C00628 V=800.0 PL=0
MOVL C00629 V=800.0 PL=0
MOVL C00630 V=800.0 PL=0
MOVL C00631 V=800.0 PL=0
MOVL C00632 V=800.0 PL=0
MOVL C00633 V=800.0 PL=0
MOVL C00634 V=800.0 PL=0
MOVL C00635 V=800.0 PL=0
MOVL C00636 V=800.0 PL=0
MOVL C00637 V=800.0 PL=0
MOVL C00638 V=800.0 PL=0
MOVL C00639 V=800.0 PL=0
MOVL C00640 V=800.0 PL=0
MOVL C00641 V=800.0 PL=0
MOVL C00642 V=800.0 PL=0
MOVL C00643 V=800.0 PL=0
MOVL C00644 V=800.0 PL=0
MOVL C00645 V=800.0 PL=0
MOVL C00646 V=800.0 PL=0
MOVL C00647 V=800.0 PL=0
MOVL C00648 V=800.0 PL=0
MOVL C00649 V=800.0 PL=0
MOVL C00650 V=800.0 PL=0
MOVL C00651 V=800.0 PL=0
MOVL C00652 V=800.0 PL=0
MOVL C00653 V=800.0 PL=0
MOVL C00654 V=800.0 PL=0
MOVL C00655 V=800.0 PL=0
MOVL C00656 V=800.0 PL=0
MOVL C00657 V=800.0 PL=0
MOVL C00658 V=800.0 PL=0
MOVL C00659 V=800.0 PL=0
MOVL C00660 V=800.0 PL=0
MOVL C00661 V=800.0 PL=0
MOVL C00662 V=800.0 PL=0
MOVL C00663 V=800.0 PL=0
MOVL C00664 V=800.0 PL=0
MOVL C00665 V=800.0 PL=0
MOVL C00666 V=800.0 PL=0
MOVL C00667 V=800.0 PL=0
MOVL C00668 V=800.0 PL=0
MOVL C00669 V=800.0 PL=0
MOVL C00670 V=800.0 PL=0
MOVL C00671 V=800.0 PL=0
MOVL C00672 V=800.0 PL=0
MOVL C00673 V=800.0 PL=0
MOVL C00674 V=800.0 PL=0
MOVL C00675 V=800.0 PL=0
MOVL C00676 V=800.0 PL=0
MOVL C00677 V=800.0 PL=0
MOVL C00678 V=800.0 PL=0
MOVL C00679 V=800.0 PL=0
MOVL C00680 V=800.0 PL=0
MOVL C00681 V=800.0 PL=0
MOVL C00682 V=800.0 PL=0
MOVL C00683 V=800.0 PL=0
MOVL C00684 V=800.0 PL=0
MOVL C00685 V=800.0 PL=0
MOVL C00686 V=800.0 PL=0
MOVL C00687 V=800.0 PL=0
MOVL C00688 V=800.0 PL=0
MOVL C00689 V=800.0 PL=0
MOVL C00690 V=800.0 PL=0
MOVL C00691 V=800.0 PL=0
MOVL C00692 V=800.0 PL=0
MOVL C00693 V=800.0 PL=0
MOVL C00694 V=800.0 PL=0
MOVL C00695 V=800.0 PL=0
MOVL C00696 V=800.0 PL=0
MOVL C00697 V=800.0 PL=0
MOVL C00698 V=800.0 PL=0
MOVL C00699 V=800.0 PL=0
MOVL C00700 V=800.0 PL=0
MOVL C00701 V=800.0 PL=0
MOVL C00702 V=800.0 PL=0
MOVL C00703 V=800.0 PL=0
MOVL C00704 V=800.0 PL=0
MOVL C00705 V=800.0 PL=0
MOVL C00706 V=800.0 PL=0
MOVL C00707 V=800.0 PL=0
MOVL C00708 V=800.0 PL=0
MOVL C00709 V=800.0 PL=0
MOVL C00710 V=800.0 PL=0
MOVL C00711 V=800.0 PL=0
MOVL C00712 V=800.0 PL=0
MOVL C00713 V=800.0 PL=0
MOVL C00714 V=800.0 PL=0
MOVL C00715 V=800.0 PL=0
MOVL C00716 V=800.0 PL=0
MOVL C00717 V=800.0 PL=0
MOVL C00718 V=800.0 PL=0
MOVL C00719 V=800.0 PL=0
MOVL C00720 V=800.0 PL=0
MOVL C00721 V=800.0 PL=0
MOVL C00722 V=800.0 PL=0
MOVL C00723 V=800.0 PL=0
MOVL C00724 V=800.0 PL=0
MOVL C00725 V=800.0 PL=0
MOVL C00726 V=800.0 PL=0
MOVL C00727 V=800.0 PL=0
MOVL C00728 V=800.0 PL=0
MOVL C00729 V=800.0 PL=0
MOVL C00730 V=800.0 PL=0
MOVL C00731 V=800.0 PL=0
MOVL C00732 V=800.0 PL=0
MOVL C00733 V=800.0 PL=0
MOVL C00734 V=800.0 PL=0
MOVL C00735 V=800.0 PL=0
MOVL C00736 V=800.0 PL=0
MOVL C00737 V=800.0 PL=0
MOVL C00738 V=800.0 PL=0
MOVL C00739 V=800.0 PL=0
MOVL C00740 V=800.0 PL=0
MOVL C00741 V=800.0 PL=0
MOVL C00742 V=800.0 PL=0
MOVL C00743 V=800.0 PL=0
MOVL C00744 V=800.0 PL=0
MOVL C00745 V=800.0 PL=0
MOVL C00746 V=800.0 PL=0
MOVL C00747 V=800.0 PL=0
MOVL C00748 V=800.0 PL=0
MOVL C00749 V=800.0 PL=0
MOVL C00750 V=800.0 PL=0
MOVL C00751 V=800.0 PL=0
MOVL C00752 V=800.0 PL=0
MOVL C00753 V=800.0 PL=0
MOVL C00754 V=800.0 PL=0
MOVL C00755 V=800.0 PL=0
MOVL C00756 V=800.0 PL=0
MOVL C00757 V=800.0 PL=0
MOVL C00758 V=800.0 PL=0
MOVL C00759 V=800.0 PL=0
MOVL C00760 V=800.0 PL=0
MOVL C00761 V=800.0 PL=0
MOVL C00762 V=800.0 PL=0
MOVL C00763 V=800.0 PL=0
MOVL C00764 V=800.0 PL=0
MOVL C00765 V=800.0 PL=0
MOVL C00766 V=800.0 PL=0
MOVL C00767 V=800.0 PL=0
MOVL C00768 V=800.0 PL=0
MOVL C00769 V=800.0 PL=0
MOVL C00770 V=800.0 PL=0
MOVL C00771 V=800.0 PL=0
MOVL C00772 V=800.0 PL=0
MOVL C00773 V=800.0 PL=0
MOVL C00774 V=800.0 PL=0
MOVL C00775 V=800.0 PL=0
MOVL C00776 V=800.0 PL=0
MOVL C00777 V=800.0 PL=0
MOVL C00778 V=800.0 PL=0
MOVL C00779 V=800.0 PL=0
MOVL C00780 V=800.0 PL=0
MOVL C00781 V=800.0 PL=0
MOVL C00782 V=800.0 PL=0
MOVL C00783 V=800.0 PL=0
MOVL C00784 V=800.0 PL=0
MOVL C00785 V=800.0 PL=0
MOVL C00786 V=800.0 PL=0
MOVL C00787 V=800.0 PL=0
MOVL C00788 V=800.0 PL=0
MOVL C00789 V=800.0 PL=0
MOVL C00790 V=800.0 PL=0
MOVL C00791 V=800.0 PL=0
MOVL C00792 V=800.0 PL=0
MOVL C00793 V=800.0 PL=0
MOVL C00794 V=800.0 PL=0
MOVL C00795 V=800.0 PL=0
MOVL C00796 V=800.0 PL=0
MOVL C00797 V=800.0 PL=0
MOVL C00798 V=800.0 PL=0
MOVL C00799 V=800.0 PL=0
MOVL C00800 V=800.0 PL=0
MOVL C00801 V=800.0 PL=0
MOVL C00802 V=800.0 PL=0
MOVL C00803 V=800.0 PL=0
MOVL C00804 V=800.0 PL=0
MOVL C00805 V=800.0 PL=0
MOVL C00806 V=800.0 PL=0
MOVL C00807 V=800.0 PL=0
MOVL C00808 V=800.0 PL=0
MOVL C00809 V=800.0 PL=0
MOVL C00810 V=800.0 PL=0
MOVL C00811 V=800.0 PL=0
MOVL C00812 V=800.0 PL=0
MOVL C00813 V=800.0 PL=0
MOVL C00814 V=800.0 PL=0
MOVL C00815 V=800.0 PL=0
MOVL C00816 V=800.0 PL=0
MOVL C00817 V=800.0 PL=0
MOVL C00818 V=800.0 PL=0
MOVL C00819 V=800.0 PL=0
MOVL C00820 V=800.0 PL=0
MOVL C00821 V=800.0 PL=0
MOVL C00822 V=800.0 PL=0
MOVL C00823 V=800.0 PL=0
MOVL C00824 V=800.0 PL=0
MOVL C00825 V=800.0 PL=0
MOVL C00826 V=800.0 PL=0
MOVL C00827 V=800.0 PL=0
MOVL C00828 V=800.0 PL=0
MOVL C00829 V=800.0 PL=0
MOVL C00830 V=800.0 PL=0
MOVL C00831 V=800.0 PL=0
MOVL C00832 V=800.0 PL=0
MOVL C00833 V=800.0 PL=0
MOVL C00834 V=800.0 PL=0
MOVL C00835 V=800.0 PL=0
MOVL C00836 V=800.0 PL=0
MOVL C00837 V=800.0 PL=0
MOVL C00838 V=800.0 PL=0
MOVL C00839 V=800.0 PL=0
MOVL C00840 V=800.0 PL=0
MOVL C00841 V=800.0 PL=0
MOVL C00842 V=800.0 PL=0
MOVL C00843 V=800.0 PL=0
MOVL C00844 V=800.0 PL=0
MOVL C00845 V=800.0 PL=0
MOVL C00846 V=800.0 PL=0
MOVL C00847 V=800.0 PL=0
MOVL C00848 V=800.0 PL=0
MOVL C00849 V=800.0 PL=0
MOVL C00850 V=800.0 PL=0
MOVL C00851 V=800.0 PL=0
MOVL C00852 V=800.0 PL=0
MOVL C00853 V=800.0 PL=0
MOVL C00854 V=800.0 PL=0
MOVL C00855 V=800.0 PL=0
MOVL C00856 V=800.0 PL=0
MOVL C00857 V=800.0 PL=0
MOVL C00858 V=800.0 PL=0
MOVL C00859 V=800.0 PL=0
MOVL C00860 V=800.0 PL=0
MOVL C00861 V=800.0 PL=0
MOVL C00862 V=800.0 PL=0
MOVL C00863 V=800.0 PL=0
MOVL C00864 V=800.0 PL=0
MOVL C00865 V=800.0 PL=0
MOVL C00866 V=800.0 PL=0
MOVL C00867 V=800.0 PL=0
MOVL C00868 V=800.0 PL=0
MOVL C00869 V=800.0 PL=0
MOVL C00870 V=800.0 PL=0
MOVL C00871 V=800.0 PL=0
MOVL C00872 V=800.0 PL=0
MOVL C00873 V=800.0 PL=0
MOVL C00874 V=800.0 PL=0
MOVL C00875 V=800.0 PL=0
MOVL C00876 V=800.0 PL=0
MOVL C00877 V=800.0 PL=0
MOVL C00878 V=800.0 PL=0
MOVL C00879 V=800.0 PL=0
MOVL C00880 V=800.0 PL=0
MOVL C00881 V=800.0 PL=0
MOVL C00882 V=800.0 PL=0
MOVL C00883 V=800.0 PL=0
MOVL C00884 V=800.0 PL=0
MOVL C00885 V=800.0 PL=0
MOVL C00886 V=800.0 PL=0
MOVL C00887 V=800.0 PL=0
MOVL C00888 V=800.0 PL=0
MOVL C00889 V=800.0 PL=0
MOVL C00890 V=800.0 PL=0
MOVL C00891 V=800.0 PL=0
MOVL C00892 V=800.0 PL=0
MOVL C00893 V=800.0 PL=0
MOVL C00894 V=800.0 PL=0
MOVL C00895 V=800.0 PL=0
MOVL C00896 V=800.0 PL=0
MOVL C00897 V=800.0 PL=0
MOVL C00898 V=800.0 PL=0
MOVL C00899 V=800.0 PL=0
MOVL C00900 V=800.0 PL=0
MOVL C00901 V=800.0 PL=0
MOVL C00902 V=800.0 PL=0
MOVL C00903 V=800.0 PL=0
MOVL C00904 V=800.0 PL=0
MOVL C00905 V=800.0 PL=0
MOVL C00906 V=800.0 PL=0
MOVL C00907 V=800.0 PL=0
MOVL C00908 V=800.0 PL=0
MOVL C00909 V=800.0 PL=0
MOVL C00910 V=800.0 PL=0
MOVL C00911 V=800.0 PL=0
MOVL C00912 V=800.0 PL=0
MOVL C00913 V=800.0 PL=0
MOVL C00914 V=800.0 PL=0
MOVL C00915 V=800.0 PL=0
MOVL C00916 V=800.0 PL=0
MOVL C00917 V=800.0 PL=0
MOVL C00918 V=800.0 PL=0
MOVL C00919 V=800.0 PL=0
MOVL C00920 V=800.0 PL=0
MOVL C00921 V=800.0 PL=0
MOVL C00922 V=800.0 PL=0
MOVL C00923 V=800.0 PL=0
MOVL C00924 V=800.0 PL=0
MOVL C00925 V=800.0 PL=0
MOVL C00926 V=800.0 PL=0
MOVL C00927 V=800.0 PL=0
MOVL C00928 V=800.0 PL=0
MOVL C00929 V=800.0 PL=0
MOVL C00930 V=800.0 PL=0
MOVL C00931 V=800.0 PL=0
MOVL C00932 V=800.0 PL=0
MOVL C00933 V=800.0 PL=0
MOVL C00934 V=800.0 PL=0
MOVL C00935 V=800.0 PL=0
MOVL C00936 V=800.0 PL=0
MOVL C00937 V=800.0 PL=0
MOVL C00938 V=800.0 PL=0
MOVL C00939 V=800.0 PL=0
MOVL C00940 V=800.0 PL=0
MOVL C00941 V=800.0 PL=0
MOVL C00942 V=800.0 PL=0
MOVL C00943 V=800.0 PL=0
MOVL C00944 V=800.0 PL=0
MOVL C00945 V=800.0 PL=0
MOVL C00946 V=800.0 PL=0
MOVL C00947 V=800.0 PL=0
MOVL C00948 V=800.0 PL=0
MOVL C00949 V=800.0 PL=0
MOVL C00950 V=800.0 PL=0
MOVL C00951 V=800.0 PL=0
MOVL C00952 V=800.0 PL=0
MOVL C00953 V=800.0 PL=0
MOVL C00954 V=800.0 PL=0
MOVL C00955 V=800.0 PL=0
MOVL C00956 V=800.0 PL=0
MOVL C00957 V=800.0 PL=0
MOVL C00958 V=800.0 PL=0
MOVL C00959 V=800.0 PL=0
MOVL C00960 V=800.0 PL=0
MOVL C00961 V=800.0 PL=0
MOVL C00962 V=800.0 PL=0
MOVL C00963 V=800.0 PL=0
MOVL C00964 V=800.0 PL=0
MOVL C00965 V=800.0 PL=0
MOVL C00966 V=800.0 PL=0
MOVL C00967 V=800.0 PL=0
MOVL C00968 V=800.0 PL=0
MOVL C00969 V=800.0 PL=0
MOVL C00970 V=800.0 PL=0
MOVL C00971 V=800.0 PL=0
MOVL C00972 V=800.0 PL=0
MOVL C00973 V=800.0 PL=0
MOVL C00974 V=800.0 PL=0
MOVL C00975 V=800.0 PL=0
MOVL C00976 V=800.0 PL=0
MOVL C00977 V=800.0 PL=0
MOVL C00978 V=800.0 PL=0
MOVL C00979 V=800.0 PL=0
MOVL C00980 V=800.0 PL=0
MOVL C00981 V=800.0 PL=0
MOVL C00982 V=800.0 PL=0
MOVL C00983 V=800.0 PL=0
MOVL C00984 V=800.0 PL=0
MOVL C00985 V=800.0 PL=0
MOVL C00986 V=800.0 PL=0
MOVL C00987 V=800.0 PL=0
MOVL C00988 V=800.0 PL=0
MOVL C00989 V=800.0 PL=0
MOVL C00990 V=800.0 PL=0
MOVL C00991 V=800.0 PL=0
MOVL C00992 V=800.0 PL=0
MOVL C00993 V=800.0 PL=0
MOVL C00994 V=800.0 PL=0
MOVL C00995 V=800.0 PL=0
MOVL C00996 V=800.0 PL=0
MOVL C00997 V=800.0 PL=0
MOVL C00998 V=800.0 PL=0
MOVL C00999 V=800.0 PL=0
MOVL C01000 V=800.0 PL=0
MOVL C01001 V=800.0 PL=0
MOVL C01002 V=800.0 PL=0
MOVL C01003 V=800.0 PL=0
MOVL C01004 V=800.0 PL=0
MOVL C01005 V=800.0 PL=0
MOVL C01006 V=800.0 PL=0
MOVL C01007 V=800.0 PL=0
MOVL C01008 V=800.0 PL=0
MOVL C01009 V=800.0 PL=0
MOVL C01010 V=800.0 PL=0
MOVL C01011 V=800.0 PL=0
MOVL C01012 V=800.0 PL=0
MOVL C01013 V=800.0 PL=0
MOVL C01014 V=800.0 PL=0
MOVL C01015 V=800.0 PL=0
MOVL C01016 V=800.0 PL=0
MOVL C01017 V=800.0 PL=0
MOVL C01018 V=800.0 PL=0
MOVL C01019 V=800.0 PL=0
MOVL C01020 V=800.0 PL=0
MOVL C01021 V=800.0 PL=0
MOVL C01022 V=800.0 PL=0
MOVL C01023 V=800.0 PL=0
MOVL C01024 V=800.0 PL=0
MOVL C01025 V=800.0 PL=0
MOVL C01026 V=800.0 PL=0
MOVL C01027 V=800.0 PL=0
MOVL C01028 V=800.0 PL=0
MOVL C01029 V=800.0 PL=0
MOVL C01030 V=800.0 PL=0
MOVL C01031 V=800.0 PL=0
MOVL C01032 V=800.0 PL=0
MOVL C01033 V=800.0 PL=0
MOVL C01034 V=800.0 PL=0
MOVL C01035 V=800.0 PL=0
MOVL C01036 V=800.0 PL=0
MOVL C01037 V=800.0 PL=0
MOVL C01038 V=800.0 PL=0
MOVL C01039 V=800.0 PL=0
MOVL C01040 V=800.0 PL=0
MOVL C01041 V=800.0 PL=0
MOVL C01042 V=800.0 PL=0
MOVL C01043 V=800.0 PL=0
MOVL C01044 V=800.0 PL=0
MOVL C01045 V=800.0 PL=0
MOVL C01046 V=800.0 PL=0
MOVL C01047 V=800.0 PL=0
MOVL C01048 V=800.0 PL=0
MOVL C01049 V=800.0 PL=0
MOVL C01050 V=800.0 PL=0
MOVL C01051 V=800.0 PL=0
MOVL C01052 V=800.0 PL=0
MOVL C01053 V=800.0 PL=0
MOVL C01054 V=800.0 PL=0
MOVL C01055 V=800.0 PL=0
MOVL C01056 V=800.0 PL=0
MOVL C01057 V=800.0 PL=0
MOVL C01058 V=800.0 PL=0
MOVL C01059 V=800.0 PL=0
MOVL C01060 V=800.0 PL=0
MOVL C01061 V=800.0 PL=0
MOVL C01062 V=800.0 PL=0
MOVL C01063 V=800.0 PL=0
MOVL C01064 V=800.0 PL=0
MOVL C01065 V=800.0 PL=0
MOVL C01066 V=800.0 PL=0
MOVL C01067 V=800.0 PL=0
MOVL C01068 V=800.0 PL=0
MOVL C01069 V=800.0 PL=0
MOVL C01070 V=800.0 PL=0
MOVL C01071 V=800.0 PL=0
MOVL C01072 V=800.0 PL=0
MOVL C01073 V=800.0 PL=0
MOVL C01074 V=800.0 PL=0
MOVL C01075 V=800.0 PL=0
MOVL C01076 V=800.0 PL=0
MOVL C01077 V=800.0 PL=0
MOVL C01078 V=800.0 PL=0
MOVL C01079 V=800.0 PL=0
MOVL C01080 V=800.0 PL=0
MOVL C01081 V=800.0 PL=0
MOVL C01082 V=800.0 PL=0
MOVL C01083 V=800.0 PL=0
MOVL C01084 V=800.0 PL=0
MOVL C01085 V=800.0 PL=0
MOVL C01086 V=800.0 PL=0
MOVL C01087 V=800.0 PL=0
MOVL C01088 V=800.0 PL=0
MOVL C01089 V=800.0 PL=0
MOVL C01090 V=800.0 PL=0
MOVL C01091 V=800.0 PL=0
MOVL C01092 V=800.0 PL=0
MOVL C01093 V=800.0 PL=0
MOVL C01094 V=800.0 PL=0
MOVL C01095 V=800.0 PL=0
MOVL C01096 V=800.0 PL=0
MOVL C01097 V=800.0 PL=0
MOVL C01098 V=800.0 PL=0
MOVL C01099 V=800.0 PL=0
MOVL C01100 V=800.0 PL=0
MOVL C01101 V=800.0 PL=0
MOVL C01102 V=800.0 PL=0
MOVL C01103 V=800.0 PL=0
MOVL C01104 V=800.0 PL=0
MOVL C01105 V=800.0 PL=0
MOVL C01106 V=800.0 PL=0
MOVL C01107 V=800.0 PL=0
MOVL C01108 V=800.0 PL=0
MOVL C01109 V=800.0 PL=0
MOVL C01110 V=800.0 PL=0
MOVL C01111 V=800.0 PL=0
MOVL C01112 V=800.0 PL=0
MOVL C01113 V=800.0 PL=0
MOVL C01114 V=800.0 PL=0
MOVL C01115 V=800.0 PL=0
MOVL C01116 V=800.0 PL=0
MOVL C01117 V=800.0 PL=0
MOVL C01118 V=800.0 PL=0
MOVL C01119 V=800.0 PL=0
MOVL C01120 V=800.0 PL=0
MOVL C01121 V=800.0 PL=0
MOVL C01122 V=800.0 PL=0
MOVL C01123 V=800.0 PL=0
MOVL C01124 V=800.0 PL=0
MOVL C01125 V=800.0 PL=0
MOVL C01126 V=800.0 PL=0
MOVL C01127 V=800.0 PL=0
MOVL C01128 V=800.0 PL=0
MOVL C01129 V=800.0 PL=0
MOVL C01130 V=800.0 PL=0
MOVL C01131 V=800.0 PL=0
MOVL C01132 V=800.0 PL=0
MOVL C01133 V=800.0 PL=0
MOVL C01134 V=800.0 PL=0
MOVL C01135 V=800.0 PL=0
MOVL C01136 V=800.0 PL=0
MOVL C01137 V=800.0 PL=0
MOVL C01138 V=800.0 PL=0
MOVL C01139 V=800.0 PL=0
MOVL C01140 V=800.0 PL=0
MOVL C01141 V=800.0 PL=0
MOVL C01142 V=800.0 PL=0
MOVL C01143 V=800.0 PL=0
MOVL C01144 V=800.0 PL=0
MOVL C01145 V=800.0 PL=0
MOVL C01146 V=800.0 PL=0
MOVL C01147 V=800.0 PL=0
MOVL C01148 V=800.0 PL=0
MOVL C01149 V=800.0 PL=0
MOVL C01150 V=800.0 PL=0
MOVL C01151 V=800.0 PL=0
MOVL C01152 V=800.0 PL=0
MOVL C01153 V=800.0 PL=0
MOVL C01154 V=800.0 PL=0
MOVL C01155 V=800.0 PL=0
MOVL C01156 V=800.0 PL=0
MOVL C01157 V=800.0 PL=0
MOVL C01158 V=800.0 PL=0
MOVL C01159 V=800.0 PL=0
MOVL C01160 V=800.0 PL=0
MOVL C01161 V=800.0 PL=0
MOVL C01162 V=800.0 PL=0
MOVL C01163 V=800.0 PL=0
MOVL C01164 V=800.0 PL=0
MOVL C01165 V=800.0 PL=0
MOVL C01166 V=800.0 PL=0
MOVL C01167 V=800.0 PL=0
MOVL C01168 V=800.0 PL=0
MOVL C01169 V=800.0 PL=0
MOVL C01170 V=800.0 PL=0
MOVL C01171 V=800.0 PL=0
MOVL C01172 V=800.0 PL=0
MOVL C01173 V=800.0 PL=0
MOVL C01174 V=800.0 PL=0
MOVL C01175 V=800.0 PL=0
MOVL C01176 V=800.0 PL=0
MOVL C01177 V=800.0 PL=0
MOVL C01178 V=800.0 PL=0
MOVL C01179 V=800.0 PL=0
MOVL C01180 V=800.0 PL=0
MOVL C01181 V=800.0 PL=0
MOVL C01182 V=800.0 PL=0
MOVL C01183 V=800.0 PL=0
MOVL C01184 V=800.0 PL=0
MOVL C01185 V=800.0 PL=0
MOVL C01186 V=800.0 PL=0
MOVL C01187 V=800.0 PL=0
MOVL C01188 V=800.0 PL=0
MOVL C01189 V=800.0 PL=0
MOVL C01190 V=800.0 PL=0
MOVL C01191 V=800.0 PL=0
MOVL C01192 V=800.0 PL=0
MOVL C01193 V=800.0 PL=0
MOVL C01194 V=800.0 PL=0
MOVL C01195 V=800.0 PL=0
MOVL C01196 V=800.0 PL=0
MOVL C01197 V=800.0 PL=0
MOVL C01198 V=800.0 PL=0
MOVL C01199 V=800.0 PL=0
MOVL C01200 V=800.0 PL=0
MOVL C01201 V=800.0 PL=0
MOVL C01202 V=800.0 PL=0
MOVL C01203 V=800.0 PL=0
MOVL C01204 V=800.0 PL=0
MOVL C01205 V=800.0 PL=0
MOVL C01206 V=800.0 PL=0
MOVL C01207 V=800.0 PL=0
MOVL C01208 V=800.0 PL=0
MOVL C01209 V=800.0 PL=0
MOVL C01210 V=800.0 PL=0
MOVL C01211 V=800.0 PL=0
MOVL C01212 V=800.0 PL=0
MOVL C01213 V=800.0 PL=0
MOVL C01214 V=800.0 PL=0
MOVL C01215 V=800.0 PL=0
MOVL C01216 V=800.0 PL=0
MOVL C01217 V=800.0 PL=0
MOVL C01218 V=800.0 PL=0
MOVL C01219 V=800.0 PL=0
MOVL C01220 V=800.0 PL=0
MOVL C01221 V=800.0 PL=0
MOVL C01222 V=800.0 PL=0
MOVL C01223 V=800.0 PL=0
MOVL C01224 V=800.0 PL=0
MOVL C01225 V=800.0 PL=0
MOVL C01226 V=800.0 PL=0
MOVL C01227 V=800.0 PL=0
MOVL C01228 V=800.0 PL=0
MOVL C01229 V=800.0 PL=0
MOVL C01230 V=800.0 PL=0
MOVL C01231 V=800.0 PL=0
MOVL C01232 V=800.0 PL=0
MOVL C01233 V=800.0 PL=0
MOVL C01234 V=800.0 PL=0
MOVL C01235 V=800.0 PL=0
MOVL C01236 V=800.0 PL=0
MOVL C01237 V=800.0 PL=0
MOVL C01238 V=800.0 PL=0
MOVL C01239 V=800.0 PL=0
MOVL C01240 V=800.0 PL=0
MOVL C01241 V=800.0 PL=0
MOVL C01242 V=800.0 PL=0
MOVL C01243 V=800.0 PL=0
MOVL C01244 V=800.0 PL=0
MOVL C01245 V=800.0 PL=0
MOVL C01246 V=800.0 PL=0
MOVL C01247 V=800.0 PL=0
MOVL C01248 V=800.0 PL=0
MOVL C01249 V=800.0 PL=0
MOVL C01250 V=800.0 PL=0
MOVL C01251 V=800.0 PL=0
MOVL C01252 V=800.0 PL=0
MOVL C01253 V=800.0 PL=0
MOVL C01254 V=800.0 PL=0
MOVL C01255 V=800.0 PL=0
MOVL C01256 V=800.0 PL=0
MOVL C01257 V=800.0 PL=0
MOVL C01258 V=800.0 PL=0
MOVL C01259 V=800.0 PL=0
MOVL C01260 V=800.0 PL=0
MOVL C01261 V=800.0 PL=0
MOVL C01262 V=800.0 PL=0
MOVL C01263 V=800.0 PL=0
MOVL C01264 V=800.0 PL=0
MOVL C01265 V=800.0 PL=0
MOVL C01266 V=800.0 PL=0
MOVL C01267 V=800.0 PL=0
MOVL C01268 V=800.0 PL=0
MOVL C01269 V=800.0 PL=0
MOVL C01270 V=800.0 PL=0
MOVL C01271 V=800.0 PL=0
MOVL C01272 V=800.0 PL=0
MOVL C01273 V=800.0 PL=0
MOVL C01274 V=800.0 PL=0
MOVL C01275 V=800.0 PL=0
MOVL C01276 V=800.0 PL=0
MOVL C01277 V=800.0 PL=0
MOVL C01278 V=800.0 PL=0
MOVL C01279 V=800.0 PL=0
MOVL C01280 V=800.0 PL=0
MOVL C01281 V=800.0 PL=0
MOVL C01282 V=800.0 PL=0
MOVL C01283 V=800.0 PL=0
MOVL C01284 V=800.0 PL=0
MOVL C01285 V=800.0 PL=0
MOVL C01286 V=800.0 PL=0
MOVL C01287 V=800.0 PL=0
MOVL C01288 V=800.0 PL=0
MOVL C01289 V=800.0 PL=0
MOVL C01290 V=800.0 PL=0
MOVL C01291 V=800.0 PL=0
MOVL C01292 V=800.0 PL=0
MOVL C01293 V=800.0 PL=0
MOVL C01294 V=800.0 PL=0
MOVL C01295 V=800.0 PL=0
MOVL C01296 V=800.0 PL=0
MOVL C01297 V=800.0 PL=0
MOVL C01298 V=800.0 PL=0
MOVL C01299 V=800.0 PL=0
MOVL C01300 V=800.0 PL=0
MOVL C01301 V=800.0 PL=0
MOVL C01302 V=800.0 PL=0
MOVL C01303 V=800.0 PL=0
MOVL C01304 V=800.0 PL=0
MOVL C01305 V=800.0 PL=0
MOVL C01306 V=800.0 PL=0
MOVL C01307 V=800.0 PL=0
MOVL C01308 V=800.0 PL=0
MOVL C01309 V=800.0 PL=0
MOVL C01310 V=800.0 PL=0
MOVL C01311 V=800.0 PL=0
MOVL C01312 V=800.0 PL=0
MOVL C01313 V=800.0 PL=0
MOVL C01314 V=800.0 PL=0
MOVL C01315 V=800.0 PL=0
MOVL C01316 V=800.0 PL=0
MOVL C01317 V=800.0 PL=0
MOVL C01318 V=800.0 PL=0
MOVL C01319 V=800.0 PL=0
MOVL C01320 V=800.0 PL=0
MOVL C01321 V=800.0 PL=0
MOVL C01322 V=800.0 PL=0
MOVL C01323 V=800.0 PL=0
MOVL C01324 V=800.0 PL=0
MOVL C01325 V=800.0 PL=0
MOVL C01326 V=800.0 PL=0
MOVL C01327 V=800.0 PL=0
MOVL C01328 V=800.0 PL=0
MOVL C01329 V=800.0 PL=0
MOVL C01330 V=800.0 PL=0
MOVL C01331 V=800.0 PL=0
MOVL C01332 V=800.0 PL=0
MOVL C01333 V=800.0 PL=0
MOVL C01334 V=800.0 PL=0
MOVL C01335 V=800.0 PL=0
MOVL C01336 V=800.0 PL=0
MOVL C01337 V=800.0 PL=0
MOVL C01338 V=800.0 PL=0
MOVL C01339 V=800.0 PL=0
MOVL C01340 V=800.0 PL=0
MOVL C01341 V=800.0 PL=0
MOVL C01342 V=800.0 PL=0
MOVL C01343 V=800.0 PL=0
MOVL C01344 V=800.0 PL=0
MOVL C01345 V=800.0 PL=0
MOVL C01346 V=800.0 PL=0
MOVL C01347 V=800.0 PL=0
MOVL C01348 V=800.0 PL=0
MOVL C01349 V=800.0 PL=0
MOVL C01350 V=800.0 PL=0
MOVL C01351 V=800.0 PL=0
MOVL C01352 V=800.0 PL=0
MOVL C01353 V=800.0 PL=0
MOVL C01354 V=800.0 PL=0
MOVL C01355 V=800.0 PL=0
MOVL C01356 V=800.0 PL=0
MOVL C01357 V=800.0 PL=0
MOVL C01358 V=800.0 PL=0
MOVL C01359 V=800.0 PL=0
MOVL C01360 V=800.0 PL=0
MOVL C01361 V=800.0 PL=0
MOVL C01362 V=800.0 PL=0
MOVL C01363 V=800.0 PL=0
MOVL C01364 V=800.0 PL=0
MOVL C01365 V=800.0 PL=0
MOVL C01366 V=800.0 PL=0
MOVL C01367 V=800.0 PL=0
MOVL C01368 V=800.0 PL=0
MOVL C01369 V=800.0 PL=0
MOVL C01370 V=800.0 PL=0
MOVL C01371 V=800.0 PL=0
MOVL C01372 V=800.0 PL=0
MOVL C01373 V=800.0 PL=0
MOVL C01374 V=800.0 PL=0
MOVL C01375 V=800.0 PL=0
MOVL C01376 V=800.0 PL=0
MOVL C01377 V=800.0 PL=0
MOVL C01378 V=800.0 PL=0
MOVL C01379 V=800.0 PL=0
MOVL C01380 V=800.0 PL=0
MOVL C01381 V=800.0 PL=0
MOVL C01382 V=800.0 PL=0
MOVL C01383 V=800.0 PL=0
MOVL C01384 V=800.0 PL=0
MOVL C01385 V=800.0 PL=0
MOVL C01386 V=800.0 PL=0
MOVL C01387 V=800.0 PL=0
MOVL C01388 V=800.0 PL=0
MOVL C01389 V=800.0 PL=0
MOVL C01390 V=800.0 PL=0
MOVL C01391 V=800.0 PL=0
MOVL C01392 V=800.0 PL=0
MOVL C01393 V=800.0 PL=0
MOVL C01394 V=800.0 PL=0
MOVL C01395 V=800.0 PL=0
MOVL C01396 V=800.0 PL=0
MOVL C01397 V=800.0 PL=0
MOVL C01398 V=800.0 PL=0
MOVL C01399 V=800.0 PL=0
MOVL C01400 V=800.0 PL=0
MOVL C01401 V=800.0 PL=0
MOVL C01402 V=800.0 PL=0
MOVL C01403 V=800.0 PL=0
MOVL C01404 V=800.0 PL=0
MOVL C01405 V=800.0 PL=0
MOVL C01406 V=800.0 PL=0
MOVL C01407 V=800.0 PL=0
MOVL C01408 V=800.0 PL=0
MOVL C01409 V=800.0 PL=0
MOVL C01410 V=800.0 PL=0
MOVL C01411 V=800.0 PL=0
MOVL C01412 V=800.0 PL=0
MOVL C01413 V=800.0 PL=0
MOVL C01414 V=800.0 PL=0
MOVL C01415 V=800.0 PL=0
MOVL C01416 V=800.0 PL=0
MOVL C01417 V=800.0 PL=0
MOVL C01418 V=800.0 PL=0
MOVL C01419 V=800.0 PL=0
MOVL C01420 V=800.0 PL=0
MOVL C01421 V=800.0 PL=0
MOVL C01422 V=800.0 PL=0
MOVL C01423 V=800.0 PL=0
MOVL C01424 V=800.0 PL=0
MOVL C01425 V=800.0 PL=0
MOVL C01426 V=800.0 PL=0
MOVL C01427 V=800.0 PL=0
MOVL C01428 V=800.0 PL=0
MOVL C01429 V=800.0 PL=0
MOVL C01430 V=800.0 PL=0
MOVL C01431 V=800.0 PL=0
MOVL C01432 V=800.0 PL=0
MOVL C01433 V=800.0 PL=0
MOVL C01434 V=800.0 PL=0
MOVL C01435 V=800.0 PL=0
MOVL C01436 V=800.0 PL=0
MOVL C01437 V=800.0 PL=0
MOVL C01438 V=800.0 PL=0
MOVL C01439 V=800.0 PL=0
MOVL C01440 V=800.0 PL=0
MOVL C01441 V=800.0 PL=0
MOVL C01442 V=800.0 PL=0
MOVL C01443 V=800.0 PL=0
MOVL C01444 V=800.0 PL=0
MOVL C01445 V=800.0 PL=0
MOVL C01446 V=800.0 PL=0
MOVL C01447 V=800.0 PL=0
MOVL C01448 V=800.0 PL=0
MOVL C01449 V=800.0 PL=0
MOVL C01450 V=800.0 PL=0
MOVL C01451 V=800.0 PL=0
MOVL C01452 V=800.0 PL=0
MOVL C01453 V=800.0 PL=0
MOVL C01454 V=800.0 PL=0
MOVL C01455 V=800.0 PL=0
MOVL C01456 V=800.0 PL=0
MOVL C01457 V=800.0 PL=0
MOVL C01458 V=800.0 PL=0
MOVL C01459 V=800.0 PL=0
MOVL C01460 V=800.0 PL=0
MOVL C01461 V=800.0 PL=0
MOVL C01462 V=800.0 PL=0
MOVL C01463 V=800.0 PL=0
MOVL C01464 V=800.0 PL=0
MOVL C01465 V=800.0 PL=0
MOVL C01466 V=800.0 PL=0
MOVL C01467 V=800.0 PL=0
MOVL C01468 V=800.0 PL=0
MOVL C01469 V=800.0 PL=0
MOVL C01470 V=800.0 PL=0
MOVL C01471 V=800.0 PL=0
MOVL C01472 V=800.0 PL=0
MOVL C01473 V=800.0 PL=0
MOVL C01474 V=800.0 PL=0
MOVL C01475 V=800.0 PL=0
MOVL C01476 V=800.0 PL=0
MOVL C01477 V=800.0 PL=0
MOVL C01478 V=800.0 PL=0
MOVL C01479 V=800.0 PL=0
MOVL C01480 V=800.0 PL=0
MOVL C01481 V=800.0 PL=0
MOVL C01482 V=800.0 PL=0
MOVL C01483 V=800.0 PL=0
MOVL C01484 V=800.0 PL=0
MOVL C01485 V=800.0 PL=0
MOVL C01486 V=800.0 PL=0
MOVL C01487 V=800.0 PL=0
MOVL C01488 V=800.0 PL=0
MOVL C01489 V=800.0 PL=0
MOVL C01490 V=800.0 PL=0
MOVL C01491 V=800.0 PL=0
MOVL C01492 V=800.0 PL=0
MOVL C01493 V=800.0 PL=0
MOVL C01494 V=800.0 PL=0
MOVL C01495 V=800.0 PL=0
MOVL C01496 V=800.0 PL=0
MOVL C01497 V=800.0 PL=0
MOVL C01498 V=800.0 PL=0
MOVL C01499 V=800.0 PL=0
MOVL C01500 V=800.0 PL=0
MOVL C01501 V=800.0 PL=0
MOVL C01502 V=800.0 PL=0
MOVL C01503 V=800.0 PL=0
MOVL C01504 V=800.0 PL=0
MOVL C01505 V=800.0 PL=0
MOVL C01506 V=800.0 PL=0
MOVL C01507 V=800.0 PL=0
MOVL C01508 V=800.0 PL=0
MOVL C01509 V=800.0 PL=0
MOVL C01510 V=800.0 PL=0
MOVL C01511 V=800.0 PL=0
MOVL C01512 V=800.0 PL=0
MOVL C01513 V=800.0 PL=0
MOVL C01514 V=800.0 PL=0
MOVL C01515 V=800.0 PL=0
MOVL C01516 V=800.0 PL=0
MOVL C01517 V=800.0 PL=0
MOVL C01518 V=800.0 PL=0
MOVL C01519 V=800.0 PL=0
MOVL C01520 V=800.0 PL=0
MOVL C01521 V=800.0 PL=0
MOVL C01522 V=800.0 PL=0
MOVL C01523 V=800.0 PL=0
MOVL C01524 V=800.0 PL=0
MOVL C01525 V=800.0 PL=0
MOVL C01526 V=800.0 PL=0
MOVL C01527 V=800.0 PL=0
MOVL C01528 V=800.0 PL=0
MOVL C01529 V=800.0 PL=0
MOVL C01530 V=800.0 PL=0
MOVL C01531 V=800.0 PL=0
MOVL C01532 V=800.0 PL=0
MOVL C01533 V=800.0 PL=0
MOVL C01534 V=800.0 PL=0
MOVL C01535 V=800.0 PL=0
MOVL C01536 V=800.0 PL=0
MOVL C01537 V=800.0 PL=0
MOVL C01538 V=800.0 PL=0
MOVL C01539 V=800.0 PL=0
MOVL C01540 V=800.0 PL=0
MOVL C01541 V=800.0 PL=0
MOVL C01542 V=800.0 PL=0
MOVL C01543 V=800.0 PL=0
MOVL C01544 V=800.0 PL=0
MOVL C01545 V=800.0 PL=0
MOVL C01546 V=800.0 PL=0
MOVL C01547 V=800.0 PL=0
MOVL C01548 V=800.0 PL=0
MOVL C01549 V=800.0 PL=0
MOVL C01550 V=800.0 PL=0
MOVL C01551 V=800.0 PL=0
MOVL C01552 V=800.0 PL=0
MOVL C01553 V=800.0 PL=0
MOVL C01554 V=800.0 PL=0
MOVL C01555 V=800.0 PL=0
MOVL C01556 V=800.0 PL=0
MOVL C01557 V=800.0 PL=0
MOVL C01558 V=800.0 PL=0
MOVL C01559 V=800.0 PL=0
MOVL C01560 V=800.0 PL=0
MOVL C01561 V=800.0 PL=0
MOVL C01562 V=800.0 PL=0
MOVL C01563 V=800.0 PL=0
MOVL C01564 V=800.0 PL=0
MOVL C01565 V=800.0 PL=0
MOVL C01566 V=800.0 PL=0
MOVL C01567 V=800.0 PL=0
MOVL C01568 V=800.0 PL=0
MOVL C01569 V=800.0 PL=0
MOVL C01570 V=800.0 PL=0
MOVL C01571 V=800.0 PL=0
MOVL C01572 V=800.0 PL=0
MOVL C01573 V=800.0 PL=0
MOVL C01574 V=800.0 PL=0
MOVL C01575 V=800.0 PL=0
MOVL C01576 V=800.0 PL=0
MOVL C01577 V=800.0 PL=0
MOVL C01578 V=800.0 PL=0
MOVL C01579 V=800.0 PL=0
MOVL C01580 V=800.0 PL=0
MOVL C01581 V=800.0 PL=0
MOVL C01582 V=800.0 PL=0
MOVL C01583 V=800.0 PL=0
MOVL C01584 V=800.0 PL=0
MOVL C01585 V=800.0 PL=0
MOVL C01586 V=800.0 PL=0
MOVL C01587 V=800.0 PL=0
MOVL C01588 V=800.0 PL=0
MOVL C01589 V=800.0 PL=0
MOVL C01590 V=800.0 PL=0
MOVL C01591 V=800.0 PL=0
MOVL C01592 V=800.0 PL=0
MOVL C01593 V=800.0 PL=0
MOVL C01594 V=800.0 PL=0
MOVL C01595 V=800.0 PL=0
MOVL C01596 V=800.0 PL=0
MOVL C01597 V=800.0 PL=0
MOVL C01598 V=800.0 PL=0
MOVL C01599 V=800.0 PL=0
MOVL C01600 V=800.0 PL=0
MOVL C01601 V=800.0 PL=0
MOVL C01602 V=800.0 PL=0
MOVL C01603 V=800.0 PL=0
MOVL C01604 V=800.0 PL=0
MOVL C01605 V=800.0 PL=0
MOVL C01606 V=800.0 PL=0
MOVL C01607 V=800.0 PL=0
MOVL C01608 V=800.0 PL=0
MOVL C01609 V=800.0 PL=0
MOVL C01610 V=800.0 PL=0
MOVL C01611 V=800.0 PL=0
MOVL C01612 V=800.0 PL=0
MOVL C01613 V=800.0 PL=0
MOVL C01614 V=800.0 PL=0
MOVL C01615 V=800.0 PL=0
MOVL C01616 V=800.0 PL=0
MOVL C01617 V=800.0 PL=0
MOVL C01618 V=800.0 PL=0
MOVL C01619 V=800.0 PL=0
MOVL C01620 V=800.0 PL=0
MOVL C01621 V=800.0 PL=0
MOVL C01622 V=800.0 PL=0
MOVL C01623 V=800.0 PL=0
MOVL C01624 V=800.0 PL=0
MOVL C01625 V=800.0 PL=0
MOVL C01626 V=800.0 PL=0
MOVL C01627 V=800.0 PL=0
MOVL C01628 V=800.0 PL=0
MOVL C01629 V=800.0 PL=0
MOVL C01630 V=800.0 PL=0
MOVL C01631 V=800.0 PL=0
MOVL C01632 V=800.0 PL=0
MOVL C01633 V=800.0 PL=0
MOVL C01634 V=800.0 PL=0
MOVL C01635 V=800.0 PL=0
MOVL C01636 V=800.0 PL=0
MOVL C01637 V=800.0 PL=0
MOVL C01638 V=800.0 PL=0
MOVL C01639 V=800.0 PL=0
MOVL C01640 V=800.0 PL=0
MOVL C01641 V=800.0 PL=0
MOVL C01642 V=800.0 PL=0
MOVL C01643 V=800.0 PL=0
MOVL C01644 V=800.0 PL=0
MOVL C01645 V=800.0 PL=0
MOVL C01646 V=800.0 PL=0
MOVL C01647 V=800.0 PL=0
MOVL C01648 V=800.0 PL=0
MOVL C01649 V=800.0 PL=0
MOVL C01650 V=800.0 PL=0
MOVL C01651 V=800.0 PL=0
MOVL C01652 V=800.0 PL=0
MOVL C01653 V=800.0 PL=0
MOVL C01654 V=800.0 PL=0
MOVL C01655 V=800.0 PL=0
MOVL C01656 V=800.0 PL=0
MOVL C01657 V=800.0 PL=0
MOVL C01658 V=800.0 PL=0
MOVL C01659 V=800.0 PL=0
MOVL C01660 V=800.0 PL=0
MOVL C01661 V=800.0 PL=0
MOVL C01662 V=800.0 PL=0
MOVL C01663 V=800.0 PL=0
MOVL C01664 V=800.0 PL=0
MOVL C01665 V=800.0 PL=0
MOVL C01666 V=800.0 PL=0
MOVL C01667 V=800.0 PL=0
MOVL C01668 V=800.0 PL=0
MOVL C01669 V=800.0 PL=0
MOVL C01670 V=800.0 PL=0
MOVL C01671 V=800.0 PL=0
MOVL C01672 V=800.0 PL=0
MOVL C01673 V=800.0 PL=0
MOVL C01674 V=800.0 PL=0
MOVL C01675 V=800.0 PL=0
MOVL C01676 V=800.0 PL=0
MOVL C01677 V=800.0 PL=0
MOVL C01678 V=800.0 PL=0
MOVL C01679 V=800.0 PL=0
MOVL C01680 V=800.0 PL=0
MOVL C01681 V=800.0 PL=0
MOVL C01682 V=800.0 PL=0
MOVL C01683 V=800.0 PL=0
MOVL C01684 V=800.0 PL=0
MOVL C01685 V=800.0 PL=0
MOVL C01686 V=800.0 PL=0
MOVL C01687 V=800.0 PL=0
MOVL C01688 V=800.0 PL=0
MOVL C01689 V=800.0 PL=0
MOVL C01690 V=800.0 PL=0
MOVL C01691 V=800.0 PL=0
MOVL C01692 V=800.0 PL=0
MOVL C01693 V=800.0 PL=0
MOVL C01694 V=800.0 PL=0
MOVL C01695 V=800.0 PL=0
MOVL C01696 V=800.0 PL=0
MOVL C01697 V=800.0 PL=0
MOVL C01698 V=800.0 PL=0
MOVL C01699 V=800.0 PL=0
MOVL C01700 V=800.0 PL=0
MOVL C01701 V=800.0 PL=0
MOVL C01702 V=800.0 PL=0
MOVL C01703 V=800.0 PL=0
MOVL C01704 V=800.0 PL=0
MOVL C01705 V=800.0 PL=0
MOVL C01706 V=800.0 PL=0
MOVL C01707 V=800.0 PL=0
MOVL C01708 V=800.0 PL=0
MOVL C01709 V=800.0 PL=0
MOVL C01710 V=800.0 PL=0
MOVL C01711 V=800.0 PL=0
MOVL C01712 V=800.0 PL=0
MOVL C01713 V=800.0 PL=0
MOVL C01714 V=800.0 PL=0
MOVL C01715 V=800.0 PL=0
MOVL C01716 V=800.0 PL=0
MOVL C01717 V=800.0 PL=0
MOVL C01718 V=800.0 PL=0
MOVL C01719 V=800.0 PL=0
MOVL C01720 V=800.0 PL=0
MOVL C01721 V=800.0 PL=0
MOVL C01722 V=800.0 PL=0
MOVL C01723 V=800.0 PL=0
MOVL C01724 V=800.0 PL=0
MOVL C01725 V=800.0 PL=0
MOVL C01726 V=800.0 PL=0
MOVL C01727 V=800.0 PL=0
MOVL C01728 V=800.0 PL=0
MOVL C01729 V=800.0 PL=0
MOVL C01730 V=800.0 PL=0
MOVL C01731 V=800.0 PL=0
MOVL C01732 V=800.0 PL=0
MOVL C01733 V=800.0 PL=0
MOVL C01734 V=800.0 PL=0
MOVL C01735 V=800.0 PL=0
MOVL C01736 V=800.0 PL=0
MOVL C01737 V=800.0 PL=0
MOVL C01738 V=800.0 PL=0
MOVL C01739 V=800.0 PL=0
MOVL C01740 V=800.0 PL=0
MOVL C01741 V=800.0 PL=0
MOVL C01742 V=800.0 PL=0
MOVL C01743 V=800.0 PL=0
MOVL C01744 V=800.0 PL=0
MOVL C01745 V=800.0 PL=0
MOVL C01746 V=800.0 PL=0
MOVL C01747 V=800.0 PL=0
MOVL C01748 V=800.0 PL=0
MOVL C01749 V=800.0 PL=0
MOVL C01750 V=800.0 PL=0
MOVL C01751 V=800.0 PL=0
MOVL C01752 V=800.0 PL=0
MOVL C01753 V=800.0 PL=0
MOVL C01754 V=800.0 PL=0
MOVL C01755 V=800.0 PL=0
MOVL C01756 V=800.0 PL=0
MOVL C01757 V=800.0 PL=0
MOVL C01758 V=800.0 PL=0
MOVL C01759 V=800.0 PL=0
MOVL C01760 V=800.0 PL=0
MOVL C01761 V=800.0 PL=0
MOVL C01762 V=800.0 PL=0
MOVL C01763 V=800.0 PL=0
MOVL C01764 V=800.0 PL=0
MOVL C01765 V=800.0 PL=0
MOVL C01766 V=800.0 PL=0
MOVL C01767 V=800.0 PL=0
MOVL C01768 V=800.0 PL=0
MOVL C01769 V=800.0 PL=0
MOVL C01770 V=800.0 PL=0
MOVL C01771 V=800.0 PL=0
MOVL C01772 V=800.0 PL=0
MOVL C01773 V=800.0 PL=0
MOVL C01774 V=800.0 PL=0
MOVL C01775 V=800.0 PL=0
MOVL C01776 V=800.0 PL=0
MOVL C01777 V=800.0 PL=0
MOVL C01778 V=800.0 PL=0
MOVL C01779 V=800.0 PL=0
MOVL C01780 V=800.0 PL=0
MOVL C01781 V=800.0 PL=0
MOVL C01782 V=800.0 PL=0
MOVL C01783 V=800.0 PL=0
MOVL C01784 V=800.0 PL=0
MOVL C01785 V=800.0 PL=0
MOVL C01786 V=800.0 PL=0
MOVL C01787 V=800.0 PL=0
MOVL C01788 V=800.0 PL=0
MOVL C01789 V=800.0 PL=0
MOVL C01790 V=800.0 PL=0
MOVL C01791 V=800.0 PL=0
MOVL C01792 V=800.0 PL=0
MOVL C01793 V=800.0 PL=0
MOVL C01794 V=800.0 PL=0
MOVL C01795 V=800.0 PL=0
MOVL C01796 V=800.0 PL=0
MOVL C01797 V=800.0 PL=0
MOVL C01798 V=800.0 PL=0
MOVL C01799 V=800.0 PL=0
MOVL C01800 V=800.0 PL=0
MOVL C01801 V=800.0 PL=0
MOVL C01802 V=800.0 PL=0
MOVL C01803 V=800.0 PL=0
MOVL C01804 V=800.0 PL=0
MOVL C01805 V=800.0 PL=0
MOVL C01806 V=800.0 PL=0
MOVL C01807 V=800.0 PL=0
MOVL C01808 V=800.0 PL=0
MOVL C01809 V=800.0 PL=0
MOVL C01810 V=800.0 PL=0
MOVL C01811 V=800.0 PL=0
MOVL C01812 V=800.0 PL=0
MOVL C01813 V=800.0 PL=0
MOVL C01814 V=800.0 PL=0
MOVL C01815 V=800.0 PL=0
MOVL C01816 V=800.0 PL=0
MOVL C01817 V=800.0 PL=0
MOVL C01818 V=800.0 PL=0
MOVL C01819 V=800.0 PL=0
MOVL C01820 V=800.0 PL=0
MOVL C01821 V=800.0 PL=0
MOVL C01822 V=800.0 PL=0
MOVL C01823 V=800.0 PL=0
MOVL C01824 V=800.0 PL=0
MOVL C01825 V=800.0 PL=0
MOVL C01826 V=800.0 PL=0
MOVL C01827 V=800.0 PL=0
MOVL C01828 V=800.0 PL=0
MOVL C01829 V=800.0 PL=0
MOVL C01830 V=800.0 PL=0
MOVL C01831 V=800.0 PL=0
MOVL C01832 V=800.0 PL=0
MOVL C01833 V=800.0 PL=0
MOVL C01834 V=800.0 PL=0
MOVL C01835 V=800.0 PL=0
MOVL C01836 V=800.0 PL=0
MOVL C01837 V=800.0 PL=0
MOVL C01838 V=800.0 PL=0
MOVL C01839 V=800.0 PL=0
MOVL C01840 V=800.0 PL=0
MOVL C01841 V=800.0 PL=0
MOVL C01842 V=800.0 PL=0
MOVL C01843 V=800.0 PL=0
MOVL C01844 V=800.0 PL=0
MOVL C01845 V=800.0 PL=0
MOVL C01846 V=800.0 PL=0
MOVL C01847 V=800.0 PL=0
MOVL C01848 V=800.0 PL=0
MOVL C01849 V=800.0 PL=0
MOVL C01850 V=800.0 PL=0
MOVL C01851 V=800.0 PL=0
MOVL C01852 V=800.0 PL=0
MOVL C01853 V=800.0 PL=0
MOVL C01854 V=800.0 PL=0
MOVL C01855 V=800.0 PL=0
MOVL C01856 V=800.0 PL=0
MOVL C01857 V=800.0 PL=0
MOVL C01858 V=800.0 PL=0
MOVL C01859 V=800.0 PL=0
MOVL C01860 V=800.0 PL=0
MOVL C01861 V=800.0 PL=0
MOVL C01862 V=800.0 PL=0
MOVL C01863 V=800.0 PL=0
MOVL C01864 V=800.0 PL=0
MOVL C01865 V=800.0 PL=0
MOVL C01866 V=800.0 PL=0
MOVL C01867 V=800.0 PL=0
MOVL C01868 V=800.0 PL=0
MOVL C01869 V=800.0 PL=0
MOVL C01870 V=800.0 PL=0
MOVL C01871 V=800.0 PL=0
MOVL C01872 V=800.0 PL=0
MOVL C01873 V=800.0 PL=0
MOVL C01874 V=800.0 PL=0
MOVL C01875 V=800.0 PL=0
MOVL C01876 V=800.0 PL=0
MOVL C01877 V=800.0 PL=0
MOVL C01878 V=800.0 PL=0
MOVL C01879 V=800.0 PL=0
MOVL C01880 V=800.0 PL=0
MOVL C01881 V=800.0 PL=0
MOVL C01882 V=800.0 PL=0
MOVL C01883 V=800.0 PL=0
MOVL C01884 V=800.0 PL=0
MOVL C01885 V=800.0 PL=0
MOVL C01886 V=800.0 PL=0
MOVL C01887 V=800.0 PL=0
MOVL C01888 V=800.0 PL=0
MOVL C01889 V=800.0 PL=0
MOVL C01890 V=800.0 PL=0
MOVL C01891 V=800.0 PL=0
MOVL C01892 V=800.0 PL=0
MOVL C01893 V=800.0 PL=0
MOVL C01894 V=800.0 PL=0
MOVL C01895 V=800.0 PL=0
MOVL C01896 V=800.0 PL=0
MOVL C01897 V=800.0 PL=0
MOVL C01898 V=800.0 PL=0
MOVL C01899 V=800.0 PL=0
MOVL C01900 V=800.0 PL=0
MOVL C01901 V=800.0 PL=0
MOVL C01902 V=800.0 PL=0
MOVL C01903 V=800.0 PL=0
MOVL C01904 V=800.0 PL=0
MOVL C01905 V=800.0 PL=0
MOVL C01906 V=800.0 PL=0
MOVL C01907 V=800.0 PL=0
MOVL C01908 V=800.0 PL=0
MOVL C01909 V=800.0 PL=0
MOVL C01910 V=800.0 PL=0
MOVL C01911 V=800.0 PL=0
MOVL C01912 V=800.0 PL=0
MOVL C01913 V=800.0 PL=0
MOVL C01914 V=800.0 PL=0
MOVL C01915 V=800.0 PL=0
MOVL C01916 V=800.0 PL=0
MOVL C01917 V=800.0 PL=0
MOVL C01918 V=800.0 PL=0
MOVL C01919 V=800.0 PL=0
MOVL C01920 V=800.0 PL=0
MOVL C01921 V=800.0 PL=0
MOVL C01922 V=800.0 PL=0
MOVL C01923 V=800.0 PL=0
MOVL C01924 V=800.0 PL=0
MOVL C01925 V=800.0 PL=0
MOVL C01926 V=800.0 PL=0
MOVL C01927 V=800.0 PL=0
MOVL C01928 V=800.0 PL=0
MOVL C01929 V=800.0 PL=0
MOVL C01930 V=800.0 PL=0
MOVL C01931 V=800.0 PL=0
MOVL C01932 V=800.0 PL=0
MOVL C01933 V=800.0 PL=0
MOVL C01934 V=800.0 PL=0
MOVL C01935 V=800.0 PL=0
MOVL C01936 V=800.0 PL=0
MOVL C01937 V=800.0 PL=0
MOVL C01938 V=800.0 PL=0
MOVL C01939 V=800.0 PL=0
MOVL C01940 V=800.0 PL=0
MOVL C01941 V=800.0 PL=0
MOVL C01942 V=800.0 PL=0
MOVL C01943 V=800.0 PL=0
MOVL C01944 V=800.0 PL=0
MOVL C01945 V=800.0 PL=0
MOVL C01946 V=800.0 PL=0
MOVL C01947 V=800.0 PL=0
MOVL C01948 V=800.0 PL=0
MOVL C01949 V=800.0 PL=0
MOVL C01950 V=800.0 PL=0
MOVL C01951 V=800.0 PL=0
MOVL C01952 V=800.0 PL=0
MOVL C01953 V=800.0 PL=0
MOVL C01954 V=800.0 PL=0
MOVL C01955 V=800.0 PL=0
MOVL C01956 V=800.0 PL=0
MOVL C01957 V=800.0 PL=0
MOVL C01958 V=800.0 PL=0
MOVL C01959 V=800.0 PL=0
MOVL C01960 V=800.0 PL=0
MOVL C01961 V=800.0 PL=0
MOVL C01962 V=800.0 PL=0
MOVL C01963 V=800.0 PL=0
MOVL C01964 V=800.0 PL=0
MOVL C01965 V=800.0 PL=0
MOVL C01966 V=800.0 PL=0
MOVL C01967 V=800.0 PL=0
MOVL C01968 V=800.0 PL=0
MOVL C01969 V=800.0 PL=0
MOVL C01970 V=800.0 PL=0
MOVL C01971 V=800.0 PL=0
MOVL C01972 V=800.0 PL=0
MOVL C01973 V=800.0 PL=0
MOVL C01974 V=800.0 PL=0
MOVL C01975 V=800.0 PL=0
MOVL C01976 V=800.0 PL=0
MOVL C01977 V=800.0 PL=0
MOVL C01978 V=800.0 PL=0
MOVL C01979 V=800.0 PL=0
MOVL C01980 V=800.0 PL=0
MOVL C01981 V=800.0 PL=0
MOVL C01982 V=800.0 PL=0
MOVL C01983 V=800.0 PL=0
MOVL C01984 V=800.0 PL=0
MOVL C01985 V=800.0 PL=0
MOVL C01986 V=800.0 PL=0
MOVL C01987 V=800.0 PL=0
MOVL C01988 V=800.0 PL=0
MOVL C01989 V=800.0 PL=0
MOVL C01990 V=800.0 PL=0
MOVL C01991 V=800.0 PL=0
MOVL C01992 V=800.0 PL=0
MOVL C01993 V=800.0 PL=0
MOVL C01994 V=800.0 PL=0
MOVL C01995 V=800.0 PL=0
MOVL C01996 V=800.0 PL=0
MOVL C01997 V=800.0 PL=0
MOVL C01998 V=800.0 PL=0
MOVL C01999 V=800.0 PL=0
MOVL C02000 V=800.0 PL=0
MOVL C02001 V=800.0 PL=0
MOVL C02002 V=800.0 PL=0
MOVL C02003 V=800.0 PL=0
MOVL C02004 V=800.0 PL=0
MOVL C02005 V=800.0 PL=0
MOVL C02006 V=800.0 PL=0
MOVL C02007 V=800.0 PL=0
MOVL C02008 V=800.0 PL=0
MOVL C02009 V=800.0 PL=0
MOVL C02010 V=800.0 PL=0
MOVL C02011 V=800.0 PL=0
MOVL C02012 V=800.0 PL=0
MOVL C02013 V=800.0 PL=0
MOVL C02014 V=800.0 PL=0
MOVL C02015 V=800.0 PL=0
MOVL C02016 V=800.0 PL=0
MOVL C02017 V=800.0 PL=0
MOVL C02018 V=800.0 PL=0
MOVL C02019 V=800.0 PL=0
MOVL C02020 V=800.0 PL=0
MOVL C02021 V=800.0 PL=0
MOVL C02022 V=800.0 PL=0
MOVL C02023 V=800.0 PL=0
MOVL C02024 V=800.0 PL=0
MOVL C02025 V=800.0 PL=0
MOVL C02026 V=800.0 PL=0
MOVL C02027 V=800.0 PL=0
MOVL C02028 V=800.0 PL=0
MOVL C02029 V=800.0 PL=0
MOVL C02030 V=800.0 PL=0
MOVL C02031 V=800.0 PL=0
MOVL C02032 V=800.0 PL=0
MOVL C02033 V=800.0 PL=0
MOVL C02034 V=800.0 PL=0
MOVL C02035 V=800.0 PL=0
MOVL C02036 V=800.0 PL=0
MOVL C02037 V=800.0 PL=0
MOVL C02038 V=800.0 PL=0
MOVL C02039 V=800.0 PL=0
MOVL C02040 V=800.0 PL=0
MOVL C02041 V=800.0 PL=0
MOVL C02042 V=800.0 PL=0
MOVL C02043 V=800.0 PL=0
MOVL C02044 V=800.0 PL=0
MOVL C02045 V=800.0 PL=0
MOVL C02046 V=800.0 PL=0
MOVL C02047 V=800.0 PL=0
MOVL C02048 V=800.0 PL=0
MOVL C02049 V=800.0 PL=0
MOVL C02050 V=800.0 PL=0
MOVL C02051 V=800.0 PL=0
MOVL C02052 V=800.0 PL=0
MOVL C02053 V=800.0 PL=0
MOVL C02054 V=800.0 PL=0
MOVL C02055 V=800.0 PL=0
MOVL C02056 V=800.0 PL=0
MOVL C02057 V=800.0 PL=0
MOVL C02058 V=800.0 PL=0
MOVL C02059 V=800.0 PL=0
MOVL C02060 V=800.0 PL=0
MOVL C02061 V=800.0 PL=0
MOVL C02062 V=800.0 PL=0
MOVL C02063 V=800.0 PL=0
MOVL C02064 V=800.0 PL=0
MOVL C02065 V=800.0 PL=0
MOVL C02066 V=800.0 PL=0
MOVL C02067 V=800.0 PL=0
MOVL C02068 V=800.0 PL=0
MOVL C02069 V=800.0 PL=0
MOVL C02070 V=800.0 PL=0
MOVL C02071 V=800.0 PL=0
MOVL C02072 V=800.0 PL=0
MOVL C02073 V=800.0 PL=0
MOVL C02074 V=800.0 PL=0
MOVL C02075 V=800.0 PL=0
MOVL C02076 V=800.0 PL=0
MOVL C02077 V=800.0 PL=0
MOVL C02078 V=800.0 PL=0
MOVL C02079 V=800.0 PL=0
MOVL C02080 V=800.0 PL=0
MOVL C02081 V=800.0 PL=0
MOVL C02082 V=800.0 PL=0
MOVL C02083 V=800.0 PL=0
MOVL C02084 V=800.0 PL=0
MOVL C02085 V=800.0 PL=0
MOVL C02086 V=800.0 PL=0
MOVL C02087 V=800.0 PL=0
MOVL C02088 V=800.0 PL=0
MOVL C02089 V=800.0 PL=0
MOVL C02090 V=800.0 PL=0
MOVL C02091 V=800.0 PL=0
MOVL C02092 V=800.0 PL=0
MOVL C02093 V=800.0 PL=0
MOVL C02094 V=800.0 PL=0
MOVL C02095 V=800.0 PL=0
MOVL C02096 V=800.0 PL=0
MOVL C02097 V=800.0 PL=0
MOVL C02098 V=800.0 PL=0
MOVL C02099 V=800.0 PL=0
MOVL C02100 V=800.0 PL=0
MOVL C02101 V=800.0 PL=0
MOVL C02102 V=800.0 PL=0
MOVL C02103 V=800.0 PL=0
MOVL C02104 V=800.0 PL=0
MOVL C02105 V=800.0 PL=0
MOVL C02106 V=800.0 PL=0
MOVL C02107 V=800.0 PL=0
MOVL C02108 V=800.0 PL=0
MOVL C02109 V=800.0 PL=0
MOVL C02110 V=800.0 PL=0
MOVL C02111 V=800.0 PL=0
MOVL C02112 V=800.0 PL=0
MOVL C02113 V=800.0 PL=0
MOVL C02114 V=800.0 PL=0
MOVL C02115 V=800.0 PL=0
MOVL C02116 V=800.0 PL=0
MOVL C02117 V=800.0 PL=0
MOVL C02118 V=800.0 PL=0
MOVL C02119 V=800.0 PL=0
MOVL C02120 V=800.0 PL=0
